// ---- Data types/TPlateData.TcDUT
{attribute 'pack_mode' := '1'}
TYPE TPlateData :
STRUCT
	lrHeight					: LREAL;
	lrEdge					: LREAL;
	alrPartOnPlate			: ARRAY[0..C_MAX_NB_OF_PARTS_ON_PLATE] OF TPositionXY;
	iNbPartOnPlate			: INT;
	alrTakePlatePos			: TPositionXY;
	lrRejectCorrectionY		: LREAL;
	bUseVisionForDrop		: BOOL;
END_STRUCT
END_TYPE

// ---- Data types/TPlatePartStatus.TcDUT
TYPE TPlatePartStatus :
	(
		PPS_Undefined := 0,
		PPS_Present,
		PPS_Absent,
		PPS_BadPart
	);
END_TYPE

// ---- Data types/TPositionXY.TcDUT
{attribute 'pack_mode' := '1'}
TYPE TPositionXY :
STRUCT
	lrX		: LREAL;
	lrY		: LREAL;
END_STRUCT
END_TYPE

// ---- Data types/TPositionXYTheta.TcDUT
{attribute 'pack_mode' := '1'}
TYPE TPositionXYTheta :
STRUCT
	lrX		: LREAL;
	lrY		: LREAL;
	lrTheta	: LREAL;
END_STRUCT
END_TYPE

// ---- Data types/TProbingArea.TcDUT
TYPE TProbingArea :
	(
		PA_BeforeSharpen := 0,
		PA_AfterSharpen,
		PA_WeightCalibration,
		PA_PartLayering1Offset0,
		PA_PartLayering1Offset1,
		PA_PartLayering2Offset0,
		PA_PartLayering2Offset1,
		PA_PartLayering3Offset0,
		PA_PartLayering3Offset1,
		PA_PartLayering4Offset0,
		PA_PartLayering4Offset1,
		PA_END
	);
END_TYPE

// ---- Data types/TProbingLog.TcDUT
{attribute 'pack_mode' := '1'}
TYPE TProbingLog :
STRUCT
	bNewLog					: BOOL;
	eProbingArea				: TProbingArea;
	alrProbingPos				: ARRAY[0..1] OF LREAL;
	iProbingThreshold				: INT;
	iPreviousProbingThreshold		: INT;
END_STRUCT
END_TYPE

// ---- Data types/TprodCounter.TcDUT
{attribute 'pack_mode' := '1'}
TYPE TprodCounter :
STRUCT
	dTotal		:DWORD;
	dGood		:DWORD;
END_STRUCT
END_TYPE

// ---- Data types/TProductionCmd.TcDUT
{attribute 'pack_mode' := '1'}
TYPE TProductionCmd :
STRUCT
	TRequestSample		: TManButton;
	TAutoSampling		: TAutoSampling;
END_STRUCT
END_TYPE

// ---- Data types/TProductionLot.TcDUT
{attribute 'pack_mode' := '1'}
TYPE TProductionLot :
STRUCT
	dLotQty					: DWORD;
	dProdQty				: DWORD;
	dGoodQty				: DWORD;
	dLoadedQty				: DWORD;
	dEstimatedPartTime		: DWORD;
	dEstimatedTimeLeft		: DWORD;
	dProductionTime			: DWORD;
END_STRUCT
END_TYPE

// ---- Data types/TProductionStats.TcDUT
{attribute 'pack_mode' := '1'}
TYPE TProductionStats :
STRUCT
	rQualityRate			: REAL;
	rEfficiencyRate		: REAL;
	rAvailabilityRate		: REAL;
END_STRUCT
END_TYPE

// ---- Data types/TRejectReason.TcDUT
TYPE TRejectReason :
	(
		RR_NoReason:=0,
		RR_PearlingSusHead1,
		RR_PearlingSusHead2,
		RR_PearlingSousHead1,
		RR_PearlingSousHead2
	);
END_TYPE

// ---- Data types/TRejectStatus.TcDUT
TYPE TRejectStatus :
	(
		RS_Ready := 0,
		RS_Locked,
		RS_Empty,
		RS_OpenDrawer
	);
END_TYPE

// ---- Data types/TRobotPos.TcDUT
{attribute 'pack_mode' := '1'}
TYPE TRobotPos :
STRUCT
	X		: LREAL;
	Y		: LREAL;
	Z		: LREAL;
	Theta	: LREAL;
END_STRUCT
END_TYPE

// ---- Data types/TRunCmdBarrel.TcDUT
TYPE TRunCmdBarrel :
	(
		RCB_None,
		RCB_GiveStick,
		RCB_PrepareStick
	);
END_TYPE

// ---- Data types/TRunCmdLift.TcDUT
TYPE TRunCmdLift :
	(
		RCL_None,
		RCL_MoveToPlate,
		RCL_MoveToLoadPlate,
		RCL_MoveToOpenDrawer
	);
END_TYPE

// ---- Data types/TRunCmdLoader.TcDUT
TYPE TRunCmdLoader :
	(
		RCLo_None,
		RCLo_TakePart,
		RCLo_GivePart,
		RCLo_TakePlate,
		RCLo_GivePlate,
		RCLo_Cleaning,
		RCLo_PrepareTakePart,
		RCLo_PrepareDropPart,
		RCLo_MoveToSafe,
		RCLo_SwitchPlate,
		RCLo_EndOfRecipe,
		RCLo_ScanPlate
	);
END_TYPE

// ---- Data types/TRunCmdPearling.TcDUT
TYPE TRunCmdPearling :
	(
		RCP_None,
		RCP_Pearl,
		RCP_ChangeChuck,
		RCP_CheckSharpen
	);
END_TYPE

// ---- Data types/TRunCmdReject.TcDUT
TYPE TRunCmdReject :
	(
		RCR_None,
		RCR_OpenDrawer,
		RCR_LockDrawer,
		RCR_UnlockDrawer
	);
END_TYPE

// ---- Data types/TRunCmdSharpen.TcDUT
TYPE TRunCmdSharpen :
	(
		RCS_None,
		RCS_MoveStep
	);
END_TYPE

// ---- Data types/TRunCmdTable.TcDUT
TYPE TRunCmdTable :
	(
		RCT_None,
		RCT_TakePart,
		RCT_GivePart,
		RCT_Turn,
		RCT_Clean,
		RCT_TurnAndClean
	);
END_TYPE

// ---- Data types/TRunCmdTurnOver.TcDUT
TYPE TRunCmdTurnOver :
	(
		RCTO_None,
		RCTO_TakePart,
		RCTO_GivePart,
		RCTO_Turn
	);
END_TYPE

// ---- Data types/TRunCmdVision.TcDUT
TYPE TRunCmdVision :
	(
		RCV_None,
		RCV_GrabImage,
		RCV_AnalyseImage
	);
END_TYPE

// ---- Data types/TRunData.TcDUT
{attribute 'pack_mode' := '1'}
TYPE TRunData :
STRUCT
	sStatusBarrel			: TRunStatus;
	sStatusLift1			: TRunStatus;
	sStatusLift2			: TRunStatus;
	sStatusLoader		: TRunStatus;
	sStatusPearling		: TRunStatus;
	sStatusReject			: TRunStatus;
	sStatusSharpen		: TRunStatus;
	sStatusTable			: TRunStatus;
	sStatusTurnOver		: TRunStatus;
	sStatusVision			: TRunStatus;
	eCmdBarrel			: TRunCmdBarrel;
	eCmdLift1			: TRunCmdLift;
	eCmdLift2			: TRunCmdLift;
	eCmdLoader			: TRunCmdLoader;
	eCmdPearling		: TRunCmdPearling;
	eCmdReject			: TRunCmdReject;
	eCmdSharpen		: TRunCmdSharpen;
	eCmdTable			: TRunCmdTable;
	eCmdTurnOver		: TRunCmdTurnOver;
	eCmdVision			: TRunCmdVision;
	TDataPearling		: TRunDataPearling;
	TDataTable			: TRunDataTable;
	TDataTurnOver		: TRunDataTurnOver;
	TDataLift1			: TRunDataLift;
	TDataLift2			: TRunDataLift;
	TDataVision			: TRunDataVision;
	TDataReject			: TRunDataReject;
	TDataLoader			: TRunDataLoader;
END_STRUCT
END_TYPE

// ---- Data types/TRunDataLift.TcDUT
{attribute 'pack_mode' := '1'}
TYPE TRunDataLift :
STRUCT
	eLiftPos			: TLiftPos;
END_STRUCT
END_TYPE

// ---- Data types/TRunDataLoader.TcDUT
{attribute 'pack_mode' := '1'}
TYPE TRunDataLoader :
STRUCT
	eTaker				: TLoaderHead;
	eModule				: TLoaderModulePos;
	iLayringPos			: INT;
	iLayringOffsetPos		: INT;
	aTPartData			: ARRAY[0..1] OF TPartData;  (* TLoaderHead *)
	bPlatePresent		: BOOL;
	lrZPositionTakeGive	: LREAL;
	iScanModel			: INT;
	iCurrentScanOK		: INT;
	iCurrentScanTotal		: INT;
END_STRUCT
END_TYPE

// ---- Data types/TRunDataPearling.TcDUT
{attribute 'pack_mode' := '1'}
TYPE TRunDataPearling :
STRUCT
		abUseSpindle				: ARRAY[0..1] OF BOOL;
		sPearlingData				: TPearlingDataHead;
		iLayringPos					: INT;
		iLayringOffsetPos				: INT;
		apsPartData					: ARRAY[0..1] OF POINTER TO TPartData;
		bForceSharpenAfterPearling	: BOOL;
END_STRUCT
END_TYPE

// ---- Data types/TRunDataPlate.TcDUT
{attribute 'pack_mode' := '1'}
TYPE TRunDataPlate :
STRUCT
	ePartStatus	: TPlatePartStatus;
END_STRUCT
END_TYPE

// ---- Data types/TRunDataReject.TcDUT
{attribute 'pack_mode' := '1'}
TYPE TRunDataReject :
STRUCT
	eRejectStatus		: TRejectStatus;
END_STRUCT
END_TYPE

// ---- Data types/TRunDataTable.TcDUT
{attribute 'pack_mode' := '1'}
TYPE TRunDataTable :
STRUCT
	aTPartData						: ARRAY[0..1,0..1,0..1] OF TPartData;	(*Layering, Layering Offset, Side *)
	iGiveTakeLayeringPosition			: INT;
	iGiveTakeLayeringOffsetPosition	: INT;
	eTableSide						: TTableSide;
END_STRUCT
END_TYPE

// ---- Data types/TRunDataTurnOver.TcDUT
{attribute 'pack_mode' := '1'}
TYPE TRunDataTurnOver :
STRUCT
	aTPartData						: ARRAY[0..1] OF TPartData;
END_STRUCT
END_TYPE

// ---- Data types/TRunDataVision.TcDUT
{attribute 'pack_mode' := '1'}
TYPE TRunDataVision :
STRUCT
		iUseModel		: INT;
		iMaxModel		: INT;
		TVisionPartData	: TVisionPartData;
END_STRUCT
END_TYPE

// ---- Data types/TRunStatus.TcDUT
TYPE TRunStatus :
	(
		RS_WaitRequest,
		RS_ProcessRequest1,
		RS_ProcessRequest2,
		RS_NotRunning
	);
END_TYPE

// ---- Data types/TStationGiversTakers.TcDUT
{attribute 'pack_mode' := '1'}
TYPE TStationGiversTakers :
	STRUCT
		(* For  loader *)
		sLoaderTurnOverTakerIn		: TTaker;
		sLoaderTurnOverGiverIn		: TGiver;
		sLoaderTurnOverTakerOut		: TTaker;
		sLoaderTurnOverGiverOut		: TGiver;

		sLoaderTableTakerIn			: TTaker;
		sLoaderTableGiverIn			: TGiver;
		sLoaderTableTakerOut		: TTaker;
		sLoaderTableGiverOut			: TGiver;


		(* For pearling station *)
		sPearlingTakeFromBarrel		:TTaker;

		(* For  barrel *)
		sBarrelGiveToPearling			:TGiver;

	END_STRUCT
END_TYPE

// ---- Data types/TStationIndex.TcDUT
TYPE TStationIndex :
	(SI_LeftLoader:=0, SI_RightLoader,SI_LeftTable,SI_LeftPearling,SI_RightTable,SI_RightPearling,SI_TurnOver,SI_LeftSharpen,SI_RightSharpen,SI_LeftBarrel,SI_RightBarrel,SI_Other);
END_TYPE

// ---- Data types/TStickData.TcDUT
{attribute 'pack_mode' := '1'}
TYPE TStickData :
STRUCT
	iBarrelPos			: INT := -1;
	lrDiameter			: LREAL;
	lrOutLength			: LREAL;
	lrTotalLength			: LREAL;
END_STRUCT
END_TYPE

// ---- Data types/TStickDataMMI.TcDUT
{attribute 'pack_mode' := '1'}
TYPE TStickDataMMI :
STRUCT
	iCompenseWeight				: INT;
	lrMCRCorrectionStep			: LREAL;
	lrMA2MMFactor				: LREAL;
	lrMCRRatio					: LREAL;
END_STRUCT
END_TYPE

// ---- Data types/TStickDataMMIShared.TcDUT
{attribute 'pack_mode' := '1'}
TYPE TStickDataMMIShared :
STRUCT
	iNbOfFwBwSharpen			: INT;
	iNbOfFwBwBeforeTapeMove	: INT;
	lrSharpenSpeed				: LREAL;
	lrSharpenHeight				: LREAL;
	bRestartBeginOfArea			: BOOL;
	lrMinHoldLength				: LREAL;
	bStopOnVacuumLoss			: BOOL;
	bStopOnStickBreak			: BOOL;
	iMCRSharpenSpeed			: INT;
	iWeightTolerance				: INT;
	bStopOnWeightOutOfTolerance	: BOOL;
END_STRUCT
END_TYPE

// ---- Data types/TStickDataShared.TcDUT
{attribute 'pack_mode' := '1'}
TYPE TStickDataShared :
STRUCT
	sStickDataMMIShared		: TStickDataMMIShared;
END_STRUCT
END_TYPE

// ---- Data types/TTableSide.TcDUT
TYPE TTableSide :
	(
		TS_A := 0,
		TS_B,
		TS_Moving
	);
END_TYPE

// ---- Data types/TTaker.TcDUT
{attribute 'pack_mode' := '1'}
TYPE TTaker :
	STRUCT
		bReadyToTake	: BOOL;		(* The taker is ready to take the part *)
		bHasTaken		: BOOL;		(* Part has been taken *)
		bHasNotTaken	: BOOL;		(* Part has not been taken *)
	END_STRUCT
END_TYPE

// ---- Data types/TTransferIndex.TcDUT
TYPE TTransferIndex :
	(TI_Loader:=0,TI_LoaderTableL1,TI_LoaderTableL2,TI_LoaderTableR1,TI_LoaderTableR2,TI_PearlingTableL,TI_PearlingTableR,TI_PearlingTable, TI_LoaderTurnOver,TI_END);
END_TYPE

// ---- Data types/TTurnOverPos.TcDUT
TYPE TTurnOverPos :
	(
		TO_Arm := 0,
		TO_Fix
	);
END_TYPE

// ---- Data types/TVaccumSettings.TcDUT
{attribute 'pack_mode' := '1'}
TYPE TVaccumSettings :
STRUCT
	iBlowing				: INT;
	iWaitWhenVacuumOk	: INT;
	iErrorDelay			: INT;
END_STRUCT
END_TYPE

// ---- Data types/TVacuumSettingsMMI.TcDUT
{attribute 'pack_mode' := '1'}
TYPE TVacuumSettingsMMI :
STRUCT
	TTable				: TVaccumSettings;
	TLoaderHead		: TVaccumSettings;
	TLoaderPlate			: TVaccumSettings;
	TTurnOver			: TVaccumSettings;
	iTablePartialDelay	: INT;
END_STRUCT
END_TYPE

// ---- Data types/TVisionData.TcDUT
{attribute 'pack_mode' := '1'}
TYPE TVisionData :
	STRUCT
		eRequest			: TVisionRequest;
		bRequestDone		: BOOL;
		bRequestError		: BOOL;
		iMajorVersion		: INT;
		iMinorVersion		: INT;
		bAlive				: BOOL;
		bConnected			: BOOL;
		acRefFileName		: STRING(20);
		TPartData			: TVisionPartData;
		bReady				: BOOL;
		bSimRecipe			: BOOL;
		iUseModel			: INT;
		iMaxModel			: INT;
		bMondemaMode		: BOOL;
		bConfigMode			: BOOL;
	END_STRUCT
END_TYPE

// ---- Data types/TVisionPartData.TcDUT
{attribute 'pack_mode' := '1'}
TYPE TVisionPartData :
	STRUCT
		lrX				: LREAL;
		lrY				: LREAL;
		lrTheta			: LREAL;
		lrScore			: LREAL;
		bValid			: BOOL;
		bPresent			: BOOL;
		bImageGrabbed	: BOOL;
	END_STRUCT
END_TYPE

// ---- Data types/TVisionRequest.TcDUT
TYPE TVisionRequest :
	(	VR_None := 0,
		VR_Init,
		VR_Analyse,
		VR_GrabImage
	);
END_TYPE

// ---- Global Variables/Global_Variables.TcGVL
{attribute 'Tc2GvlVarNames'}
(*-----------------------------------------------------------------------------------------------------------------------------------------------------------------------------------------------------------------------------------------------------------------------------------------------------------------------
  GLOBAL CONFIGURATION SPECIFIC TO SOLD MACHINE
 *)
VAR_GLOBAL PERSISTENT
	bUseMDEOption							: BOOL							:= TRUE;	(* MDE option for ETA *)
	bUseRTPOption							: BOOL							:= FALSE;	(* REAL-TIME pearling screen option *)
	bUseTurnOverOption						: BOOL							:= FALSE;	(* TurnOver module is fitted *)
	bUseASOption							: BOOL							:= FALSE;	(* Auto-Sampling screen option *)
	bUseNewBarrelFunction					: BOOL							:= TRUE;	(* Specific function to use 1-4 sectors for each gripper *)
	bUse103059Kludges						: BOOL							:= FALSE;	(* Specific to Blancpain to correct mechanical issues *)
	bRejectPartWithVacuumErrorOnTable		: BOOL							:= FALSE;	(* Try to reject a part if vacuum on table was bad when dropping from loader *)
	bUseFullTapeWidth						: BOOL							:= FALSE;	(* Use full tape width, half for roughing, other half for finish *)
	bUsePearlMoveToSafe						: BOOL							:= FALSE;	(* Use the feature to not move to preref between pearls to save time *)
	bUseLockPlate							: bool							:= False; 	(* Use the lock plate option of the Lifts *)
(* Optimisations *)
	bUse103171OptimA1						: BOOL							:= FALSE;	(* Specific optimisation specified in document 502004-3TC-0001-07 *)
	bUse103171OptimB3						: BOOL							:= FALSE;	(* Specific optimisation specified in document 502004-3TC-0001-07 *)
	bUse103171OptimB5PreMoveXY				: BOOL							:= FALSE;	(* Specific optimisation specified in document 502004-3TC-0001-07 : Pre-move XY to safe when waiting for others *)
	bUse103171OptimB5MoveOnPreSafeZ			: BOOL							:= FALSE;	(* Specific optimisation specified in document 502004-3TC-0001-07 : Say Z in safe if near by safe position even if not in position *)
	bUse103171OptimB5CleanOnBothSide		: BOOL							:= FALSE;	(* Specific optimisation specified in document 502004-3TC-0001-07 : Clean on both side *)
	bUse103171OptimB5CleanOn1Move			: BOOL							:= FALSE;	(* Specific optimisation specified in document 502004-3TC-0001-07 : Clean only on 1 move (no return back *)
END_VAR
VAR_GLOBAL CONSTANT
	C_MAX_NB_OF_ERRORS						: INT							:= 159;		(* 160 errors *)
	C_MAX_NB_OF_PARTS_ON_PLATE				: INT							:= 99;		(* Max nb of parts on plate : 100*)
	C_MAX_NB_OF_PEARLS						: INT							:= 600;		(* Max NB of pearls on 1 side and 1 diameter *)
	C_NB_OF_COM								: INT							:=1;		(* Nb of serial ports *)
	C_COM_NUMBERS							: ARRAY[1..C_NB_OF_COM] OF INT	:= [1];		(* List of serial ports com numbers *)
	C_WEIGHT_TABLE_MAX						: INT							:=25;		(* Nb of point for weight calibration *)
	C_PROD_MODE_GOOD_PART					: BOOL							:= FALSE;	(* False -> Prod quantity is the number of parts on the lift / True -> Prod quantity is the good produced part *)
END_VAR
(*-----------------------------------------------------------------------------------------------------------------------------------------------------------------------------------------------------------------------------------------------------------------------------------------------------------------------*)
VAR_GLOBAL
(* For MDE *)
	{attribute 'OPC.UA.DA' := '1'}
  	{attribute 'OPC.UA.DA.StructuredType' := '1'}
	TMDEData								: TMDE; 									(* TMDE Data *)
(* Internal data *)
	RxBuffer_MCR							: ARRAY[1..C_NB_OF_COM] OF ComBuffer;		(* Reception buffer for MCR *)
	TxBuffer_MCR							: ARRAY[1..C_NB_OF_COM] OF ComBuffer;		(* Transmission buffer for MCR *)
(* Digital IOs *)
	(* Twinsafe *)
	IbV1PowerIsOff					AT %I*	: BOOL;										(* TWINSAFE : Power V1 is off *)
	IbDrivesAreOFF					AT %I*	: BOOL;										(* TWINSAFE : Power on drives is off *)
	IbNoEmergencyStop				AT %I*	: BOOL;										(* TWINSAFE : Emergency stop not pressed *)
	QbStartSafety					AT %Q*	: BOOL;										(* TWINSAFE : Start the safety **Always set to true** *)
	QbPowerOnDrives					AT %Q*	: BOOL;										(* TWINSAFE : Power on drives **Always set to true** *)
	QbResetSafety					AT %Q*	: BOOL;										(* TWINSAFE : Reset the safety errors *)
	(* Doors *)
	IbPearlingDoorsClosed			AT %I*	: BOOL;										(* Pearling doors are closed *)
	IbPearlingDoorsLocked			AT %I*	: BOOL;										(* Pearling doors are locked *)
	IbLoaderDoorsClosed				AT %I*	: BOOL;										(* Loader doors are closed *)
	IbLoaderDoorsLocked				AT %I*	: BOOL;										(* Loader doors are locked *)
	QbLockPearlingDoors				AT %Q*	: BOOL;										(* Lock door on pearling *)
	QbLockLoaderDoors				AT %Q*	: BOOL;										(* Lock door on loader *)
	(* Power supplies *)
	Ib24VOK							AT %I*	: BOOL;										(* 24V power supplies are OK *)
	Ib48VOK							AT %I*	: BOOL;										(* 48V power supplies are OK *)
	(* Light Tower *)
	QbGreenLight					AT %Q*	: BOOL;										(* Green light *)
	QbRedLight						AT %Q*	: BOOL;										(* Red light *)
	QbBlueLight						AT %Q*	: BOOL;										(* Yellow light *)
	(*Air pressure *)
	IbAirPressureOK					AT %I*	: BOOL;										(* Air pressure is OK *)
	(* Vacuum *)
	IbVacuumPumpIsOn				AT %I*	: BOOL;										(* Vacuum pump is powered *)
	IbMainVacuumOK					AT %I*	: BOOL;										(* main vacuum is OK *)
	QbVacuumPumpOn					AT %Q*	: BOOL;										(* Activate vacuum pump *)
	(* Aspiration *)
	IbAspirationIsOn				AT %I*	: BOOL;										(* Aspiration is powered *)
	IbAspirationOK					AT %I*	: BOOL;										(* Aspiration is OK *)
	QbAspirationOn					AT %Q*	: BOOL;										(* Activate aspirator *)
	(* Lift 1 *)
	IbLift1Home						AT %I*	: BOOL;										(* Lift 1 is at home *)
	IbLift1PosLimit					AT %I*	: BOOL;										(* Lift 1 is not down *)
	IbLift1NegLimit					AT %I*	: BOOL;										(* Lift 1 is not up *)
	IbLift1PlateInPos				AT %I*	: BOOL;										(* Plate on lift 1 is in position *)
	IbLift1DrawerInPos				AT %I*	: BOOL;										(* Drawer of lift 1 is in position *)
	IbLift1DrawerLocked				AT %I*	: BOOL;										(* Drawer of lift 1 is locked *)
	IbLift1DrawerUnlocked			AT %I*	: BOOL;										(* Drawer of lift 1 is unlocked *)
	IbLift1PlateLocked				AT %I*	: BOOL;										(* Lift 1 plate is locked *)
	IbLift1PlateUnlocked			AT %I*	: BOOL;										(* Lift 1 plate is unlocked *)
	QbLift1BlueLight				AT %Q*	: BOOL;										(* Blue light for left lift *)
	QbLift1LockPlate				AT %Q*	: BOOL;										(* Lock plate of lift 1 *)
	QbLift1UnlockPlate				AT %Q*	: BOOL;										(* Unlock plate of lift 1 *)
	QbLift1LockDrawer				AT %Q*	: BOOL;										(* Lock drawer of lift 1 *)
	QbLift1UnlockDrawer				AT %Q*	: BOOL;										(* Unlock drawer of lift 1 *)
	(* Lift 2 *)
	IbLift2Home						AT %I*	: BOOL;										(* Lift 1 is at home *)
	IbLift2PosLimit					AT %I*	: BOOL;										(* Lift 2 is not down *)
	IbLift2NegLimit					AT %I*	: BOOL;										(* Lift 2 is not up *)
	IbLift2PlateInPos				AT %I*	: BOOL;										(* Plate on lift 2 is in position *)
	IbLift2DrawerInPos				AT %I*	: BOOL;										(* Drawer of lift 2 is in position *)
	IbLift2DrawerLocked				AT %I*	: BOOL;										(* Drawer of lift 2 is locked *)
	IbLift2DrawerUnlocked			AT %I*	: BOOL;										(* Drawer of lift 2 is unlocked *)
	IbLift2PlateLocked				AT %I*	: BOOL;										(* Lift 2 plate is locked *)
	IbLift2PlateUnlocked			AT %I*	: BOOL;										(* Lift 2 plate is unlocked *)
	QbLift2BlueLight				AT %Q*	: BOOL;										(* Blue light for right lift *)
	QbLift2LockPlate				AT %Q*	: BOOL;										(* Lock plate of lift 2 *)
	QbLift2UnlockPlate				AT %Q*	: BOOL;										(* Unlock plate of lift 2 *)
	QbLift2LockDrawer				AT %Q*	: BOOL;										(* Lock drawer of lift 2 *)
	QbLift2UnlockDrawer				AT %Q*	: BOOL;										(* Unlock drawer of lift 2 *)
	(* Reject *)
	IbRejectPlateInPos				AT %I*	: BOOL;										(* Plate on reject is in position *)
	IbRejectDrawerInPos				AT %I*	: BOOL;										(* Drawer for reject is in position *)
	QbRejectBlueLight				AT %Q*	: BOOL;										(* Blue light for reject *)
	(* Loader *)
	ILoaderMotorXYStatus			AT %I*	: WORD;										(* Digital inputs from loader XY drive *)
	IbLoaderHomeZ1					AT %I*	: BOOL;										(* Home for Head 1 Z axis *)
	IbLoaderPosLimitZ1				AT %I*	: BOOL;										(* Pos. llimit for Head 1 Z axis *)
	IbLoaderNegLimitZ1				AT %I*	: BOOL;										(* Neg. llimit for Head 1 Z axis *)
	IbLoaderHomeZ2					AT %I*	: BOOL;										(* Home for Head 2 Z axis *)
	IbLoaderPosLimitZ2				AT %I*	: BOOL;										(* Pos. llimit for Head 2 Z axis *)
	IbLoaderNegLimitZ2				AT %I*	: BOOL;										(* Neg. llimit for Head 2 Z axis *)
	IbLoaderPlateTakerIsUp			AT %I*	: BOOL;										(* Plate taker is up *)
	IbLoaderPlateTakerIsDown		AT %I*	: BOOL;										(* Plate taker is down *)
	IiLoaderHead1Vacuum				AT %I*	: INT;										(* Vacuum flow on head 1 *)
	IiLoaderHead2Vacuum				AT %I*	: INT;										(* Vacuum flow on head 2 *)
	IbLoaderPlateVacuumOK			AT %I*	: BOOL;										(* Vacuum on plate is OK *)
	ILoaderPlateDistance			AT %I*	: INT;										(* Distance from head to plate *)
	QbLoaderActivateHead1Vacuum		AT %Q*	: BOOL;										(* Activate Head 1 vacuum *)
	QbLoaderActivateHead1Blowing	AT %Q*	: BOOL;										(* Activate Head 1 blowing *)
	QbLoaderActivateHead2Vacuum		AT %Q*	: BOOL;										(* Activate Head 2 vacuum *)
	QbLoaderActivateHead2Blowing	AT %Q*	: BOOL;										(* Activate Head 2 blowing *)
	QbLoaderActivatePlateVacuum		AT %Q*	: BOOL;										(* Activate plate vacuum *)
	QbLoaderActivatePlateBlowing	AT %Q*	: BOOL;										(* Activate plate blowing *)
	QbLoaderPlateTakerDown			AT %Q*	: BOOL;										(* Move down the plate taker part *)
	QbLoaderPlateTakerUp			AT %Q*	: BOOL;										(* Move up the plate taker part *)
	QbLoaderBrushAspirationVacuum	AT %Q*	: BOOL;										(* Activate aspiration on cleaning brush *)
	QbLoaderBrushAspirationBlowing	AT %Q*	: BOOL;										(* Deactivate aspiration on cleaning brush *)
	(* Table *)
	IbTableHome						AT %I*	: BOOL;										(* Home for rotation axis *)
	IbTableLocked					AT %I*	: BOOL;										(* Table is locked in position *)
	IbTableNotLocked				AT %I*	: BOOL;										(* Table is not locked in position *)
	IiTableVacuumPos1Flow			AT %I*	: INT;										(* Vacuum flow on position 1 *)
	IiTableVacuumPos2Flow			AT %I*	: INT;										(* Vacuum flow on position 2 *)
	IiTableVacuumPos3Flow			AT %I*	: INT;										(* Vacuum flow on position 3 *)
	IiTableVacuumPos4Flow			AT %I*	: INT;										(* Vacuum flow on position 4 *)
	IbTableAspirationIsUp			AT %I*	: BOOL;										(* Aspiration module is up *)
	IbTableAspirationIsDown			AT %I*	: BOOL;										(* Aspiration module is down *)
	IbTableCleanBrushIsUp			AT %I*	: BOOL;										(* Clean brush is up *)
	IbTableCleanBrushIsDown			AT %I*	: BOOL;										(* Clean brush is down *)
	QbTableLock						AT %Q*	: BOOL;										(* Lock the table in position *)
	QbTableActivateVacuumPos1		AT %Q*	: BOOL;										(* Activate vacuum on position 1 *)
	QbTableActivateBlowingPos1		AT %Q*	: BOOL;										(* Activate blowing on position 1 *)
	QbTableActivateVacuumPos2		AT %Q*	: BOOL;										(* Activate vacuum on position 2 *)
	QbTableActivateBlowingPos2		AT %Q*	: BOOL;										(* Activate blowing on position 2 *)
	QbTableActivateVacuumPos3		AT %Q*	: BOOL;										(* Activate vacuum on position 3 *)
	QbTableActivateBlowingPos3		AT %Q*	: BOOL;										(* Activate blowing on position 3 *)
	QbTableActivateVacuumPos4		AT %Q*	: BOOL;										(* Activate vacuum on position 4 *)
	QbTableActivateBlowingPos4		AT %Q*	: BOOL;										(* Activate blowing on position 4 *)
	QbTableAspiration13Vacuum		AT %Q*	: BOOL;										(* Activate aspiration on left position *)
	QbTableAspiration13Blowing		AT %Q*	: BOOL;										(* Activate aspiration on right position *)
	QbTableAspiration24Vacuum		AT %Q*	: BOOL;										(* Deactivate aspiration on left position *)
	QbTableAspiration24Blowing		AT %Q*	: BOOL;										(* Deactivate aspiration on right position *)
	QbTableAspirationUp				AT %Q*	: BOOL;										(* Move aspiration module down *)
	QbTableAspirationDown			AT %Q*	: BOOL;										(* Move aspiration module down *)
	QbTableCleanBrushDown			AT %Q*	: BOOL;										(* Move clean brush down *)
	(* Brush *)
	IbBrushHome						AT %I*	: BOOL;										(* Home for Brush axis *)
	IbBrushPosLimit					AT %I*	: BOOL;										(* Pos. llimit for Brush axis *)
	IbBrushNegLimit					AT %I*	: BOOL;										(* Neg limit for Brush axis *)
	QbBrushAspirationVacuum			AT %Q*	: BOOL;										(* Activate aspiration on cleaning brush *)
	QbBrushAspirationBlowing		AT %Q*	: BOOL;										(* Deactivate aspiration on cleaning brush *)
	(* Pearling *)
	IPearlingMotorXYStatus			AT %I*	: WORD;										(* Digital inputs from pearling XY drive *)
	IbPearlingHomeZ1				AT %I*	: BOOL;										(* Home for Z1 axis *)
	IbPearlingPosLimitZ1			AT %I*	: BOOL;										(* Pos. llimit for Z1 axis *)
	IbPearlingNegLimitZ1			AT %I*	: BOOL;										(* Neg. llimit for Z1 axis *)
	IbPearlingHomeZ2				AT %I*	: BOOL;										(* Home for Z2 axis *)
	IbPearlingPosLimitZ2			AT %I*	: BOOL;										(* Pos. llimit for Z2 axis *)
	IbPearlingNegLimitZ2			AT %I*	: BOOL;										(* Neg. llimit for Z2 axis *)
	IbPearlingChuck1Open			AT %I*	: BOOL;										(* Chuck 1 is open *)
	IbPearlingChuck1Closed			AT %I*	: BOOL;										(* Chuck 1 is closed *)
	IbPearlingChuck2Open			AT %I*	: BOOL;										(* Chuck 2 is open *)
	IbPearlingChuck2Closed			AT %I*	: BOOL;										(* Chuck 2 is closed *)
	IbPearlingChangeBroach			AT %I*	: BOOL;										(* Request change broach button*)
	IPearlingContact1Distance		AT %I*	: INT;										(* Distance from sensor to stick 1 contact *)
	IPearlingContact2Distance		AT %I*	: INT;										(* Distance from sensor to stick 2 contact *)
	IPearlingWeightMeasure			AT %I*	: INT;										(* Weight on load sensor *)
	QbPearlingStartMotor1			AT %Q*	: BOOL;										(* Start the pearling 1 motor *)
	QbPearlingStartMotor2			AT %Q*	: BOOL;										(* Start the pearling 2 motor *)
	QbPearlingOpenChuck1			AT %Q*	: BOOL;										(* Open chuck 1 *)
	QbPearlingOpenChuck2			AT %Q*	: BOOL;										(* Open chuck 2 *)
	QbPearlingActivateEject1		AT %Q*	: BOOL;										(* Activate stick 1 ejection *)
	QbPearlingActivateEject2		AT %Q*	: BOOL;										(* Activate stick 2 ejection *)
	QbPearlingActivateBlowing1		AT %Q*	: BOOL;										(* Activate blowing 1 *)
	QbPearlingActivateBlowing2		AT %Q*	: BOOL;										(* Activate blowing 2 *)
	QbPearlingStickLed1				AT %Q*	: BOOL;										(* Stick 1 led is on *)
	QbPearlingStickLed2				AT %Q*	: BOOL;										(* Stick 2 led is on *)
	QbPearlingChangeBroachLight		AT %Q*	: BOOL;										(* Request change broach button light*)
	(* TurnOver *)
	IbTurnOverHome					AT %I*	: BOOL;										(* Home for axis *)
	IbTurnOverArmVacuumOK			AT %I*	: BOOL;										(* Vacuum is OK on arm *)
	IbTurnOverFixVacuumOK			AT %I*	: BOOL;										(* Vacuum is OK on fix position *)
	IbTurnOverFixIsUp				AT %I*	: BOOL;										(* Fix is up *)
	IbTurnOverFixIsDown				AT %I*	: BOOL;										(* Fix is down *)
	QbTurnOverActivateVacuumArm		AT %Q*	: BOOL;										(* Activate vacuum on arm *)
	QbTurnOverActivateBlowingArm	AT %Q*	: BOOL;										(* Activate blowing on arm *)
	QbTurnOverActivateVacuumFix		AT %Q*	: BOOL;										(* Activate vacuum on fix position *)
	QbTurnOverActivateBlowingFix	AT %Q*	: BOOL;										(* Activate blowing on fix position *)
	QbTurnOverMoveFixUp				AT %Q*	: BOOL;										(* Move fix up *)
	QbTurnOverMoveFixDown			AT %Q*	: BOOL;										(* Move fix down *)
	QbTurnOverActivateCleaningBlow	AT %Q*	: BOOL;										(* Activate blowing to clean the holder *)
	(* Sharpen *)
	IbSharpenPosTensioner			AT %I*	: BOOL;										(* The sharpening band is not empty *)
	QbSharpenAspirationVacuum		AT %Q*	: BOOL;										(* Activate aspiration on sharpen*)
	QbSharpenAspirationBlowing		AT %Q*	: BOOL;										(* Deactivate aspiration on sharpen*)
	(* Barrel *)
	IbBarrelStickIsUp				AT %I*	: BOOL;										(* Stick is up *)
	IbBarrelStickIsDown				AT %I*	: BOOL;										(* Stick is down *)
	IbBarrelStickPresent			AT %I*	: BOOL;										(* A stick is present on sensor *)
	IbBarrelIndexed					AT %I*	: BOOL;										(* The barrel is indexed *)
	IbBarrelNotIndexed				AT %I*	: BOOL;										(* The barrel is not indexed *)
	QbBarrelMoveUpStick				AT %Q*	: BOOL;										(* Move up stick *)
	QbBarrelIndexTable				AT %Q*	: BOOL;										(* Move up index *)
	(* Axis *)
	TLoaderXAxis							: AXIS_REF				;					(* linked to loader X axis var in TWINCAT System Manager *)
	TLoaderYAxis							: AXIS_REF;									(* linked to loader Y axis var in TWINCAT System Manager *)
	TLoaderZ1Axis							: AXIS_REF;									(* linked to loader Head 1 Z axis var in TWINCAT System Manager *)
	TLoaderZ2Axis							: AXIS_REF;									(* linked to  loader Head 2 Z axis var in TWINCAT System Manager *)
	TLoaderThetaAxis						: AXIS_REF;									(* linked to  loader Theta axis var in TWINCAT System Manager *)
	TLift1Axis								: AXIS_REF;									(* linked to left lift axis var in TWINCAT System Manager *)
	TLift2Axis								: AXIS_REF;									(* linked to right lift axis var in TWINCAT System Manager *)
	TPearlingXAxis							: AXIS_REF;									(* linked to pearling X axis var in TWINCAT System Manager *)
	TPearlingYAxis							: AXIS_REF;									(* linked to pearling Y axis var in TWINCAT System Manager *)
	TPearlingZ1Axis							: AXIS_REF;									(* linked to pearling Z1 axis var in TWINCAT System Manager *)
	TPearlingZ2Axis							: AXIS_REF;									(* linked to pearling Z2 axis var in TWINCAT System Manager *)
	TTableAxis								: AXIS_REF;									(* linked to table axis var in TWINCAT System Manager *)
	TTurnOverAxis							: AXIS_REF;									(* linked to turn over axis var in TWINCAT System Manager *)
	TSharpenAxis							: AXIS_REF;									(* linked to sharpen axis var in TWINCAT System Manager *)
	TSharpenEncoder							: AXIS_REF;									(* linked to sharpen encoder var in TWINCAT System Manager *)
	TBarrelAxis								: AXIS_REF;									(* linked to barrel axis var in TWINCAT System Manager *)
	TBrushAxis								: AXIS_REF;									(* linked to brush axis var in TWINCAT System Manager *)
END_VAR

// ---- Global Variables/TwinCAT_Configuration.TcGVL
{attribute 'Tc2GvlVarNames'}
(* Generated automatically by TwinCAT - (read only) *)
VAR_CONFIG
	.IbV1PowerIsOff AT %IX52.2 : BOOL;	(*  ~ {LinkedWith:TIID^Device 2 (EtherCAT)^A22.A (Term IO)^A29.4 (TwinSafe IN)^Module 1 (FSOES)^TxPDO^FSOE^PwrV1IsOn_1} *)
	.IbDrivesAreOFF AT %IX52.3 : BOOL;	(*  ~ {LinkedWith:TIID^Device 2 (EtherCAT)^A22.A (Term IO)^A29.4 (TwinSafe IN)^Module 1 (FSOES)^TxPDO^FSOE^DriveIsOn1} *)
	.IbNoEmergencyStop AT %IX52.4 : BOOL;	(*  ~ {LinkedWith:TIID^Device 2 (EtherCAT)^A22.A (Term IO)^A29.1 (TwinSafe PLC)^Module 2 (FSOE)^Standard Out Vars TxPDO 1^Standard Out Var 1} *)
	.QbStartSafety AT %QX0.1 : BOOL;	(*  ~ {LinkedWith:TIID^Device 2 (EtherCAT)^A22.A (Term IO)^A29.1 (TwinSafe PLC)^Module 2 (FSOE)^Standard In Vars RxPDO 1^Standard In Var 1} *)
	.QbPowerOnDrives AT %QX1.1 : BOOL;	(*  ~ {LinkedWith:TIID^Device 2 (EtherCAT)^A22.A (Term IO)^A29.1 (TwinSafe PLC)^Module 2 (FSOE)^Standard In Vars RxPDO 1^Standard In Var 4} *)
	.QbResetSafety AT %QX0.2 : BOOL;	(*  ~ {LinkedWith:TIID^Device 2 (EtherCAT)^A22.A (Term IO)^A29.1 (TwinSafe PLC)^Module 2 (FSOE)^Standard In Vars RxPDO 1^Standard In Var 2;
													TIID^Device 2 (EtherCAT)^A22.A (Term IO)^A29.1 (TwinSafe PLC)^Module 2 (FSOE)^Standard In Vars RxPDO 1^Standard In Var 3;
													TIID^Device 2 (EtherCAT)^A22.A (Term IO)^A29.1 (TwinSafe PLC)^Module 2 (FSOE)^Standard In Vars RxPDO 1^Standard In Var 5} *)
	.IbPearlingDoorsClosed AT %IX52.5 : BOOL;	(*  ~ {LinkedWith:TIID^Device 2 (EtherCAT)^A22.A (Term IO)^A29.3 (TwinSafe IN)^Module 1 (FSOES)^TxPDO^FSOE^Safety3-4Sec1} *)
	.IbPearlingDoorsLocked AT %IX2516.0 : BOOL;	(*  ~ {LinkedWith:TIID^Device 2 (EtherCAT)^A22.A (Term IO)^A29.3 (TwinSafe IN)^Module 1 (FSOES)^TxPDO^FSOE^Safety3-4Sec2} *)
	.IbLoaderDoorsClosed AT %IX52.7 : BOOL;	(*  ~ {LinkedWith:TIID^Device 2 (EtherCAT)^A22.A (Term IO)^A29.3 (TwinSafe IN)^Module 1 (FSOES)^TxPDO^FSOE^Safety1-2Sec1} *)
	.IbLoaderDoorsLocked AT %IX2516.1 : BOOL;	(*  ~ {LinkedWith:TIID^Device 2 (EtherCAT)^A22.A (Term IO)^A29.3 (TwinSafe IN)^Module 1 (FSOES)^TxPDO^FSOE^Safety1-2Sec2} *)
	.QbLockPearlingDoors AT %QX2444.0 : BOOL;	(*  ~ {LinkedWith:TIID^Device 2 (EtherCAT)^A22.A (Term IO)^A26.1^Channel 3^Safety3Lock;TIID^Device 2 (EtherCAT)^A22.A (Term IO)^A26.1^Channel 4^Safety4Lock} *)
	.QbLockLoaderDoors AT %QX2444.1 : BOOL;	(*  ~ {LinkedWith:TIID^Device 2 (EtherCAT)^A22.A (Term IO)^A26.1^Channel 1^Safety1Lock;TIID^Device 2 (EtherCAT)^A22.A (Term IO)^A26.1^Channel 2^Safety2Lock} *)
	.Ib24VOK AT %IX52.0 : BOOL;	(*  ~ {LinkedWith:TIID^Device 2 (EtherCAT)^A22.A (Term IO)^A22.1^Channel 1^Supply24VOn} *)
	.Ib48VOK AT %IX52.1 : BOOL;	(*  ~ {LinkedWith:TIID^Device 2 (EtherCAT)^A22.A (Term IO)^A22.1^Channel 2^Supply48VOn} *)
	.QbGreenLight AT %QX0.3 : BOOL;	(*  ~ {LinkedWith:TIID^Device 2 (EtherCAT)^A22.A (Term IO)^A26.2^Channel 1^GreenLight} *)
	.QbRedLight AT %QX0.5 : BOOL;	(*  ~ {LinkedWith:TIID^Device 2 (EtherCAT)^A22.A (Term IO)^A26.2^Channel 2^RedLight} *)
	.QbBlueLight AT %QX0.4 : BOOL;	(*  ~ {LinkedWith:TIID^Device 2 (EtherCAT)^A22.A (Term IO)^A26.2^Channel 3^BlueLight} *)
	.IbAirPressureOK AT %IX53.1 : BOOL;	(*  ~ {LinkedWith:TIID^Device 2 (EtherCAT)^A22.A (Term IO)^A22.1^Channel 3^AirSupplyOk} *)
	.IbVacuumPumpIsOn AT %IX2516.2 : BOOL;	(*  ~ {LinkedWith:TIID^Device 2 (EtherCAT)^A22.A (Term IO)^A22.1^Channel 6^VacuumPumpIsOn} *)
	.IbMainVacuumOK AT %IX53.3 : BOOL;	(*  ~ {LinkedWith:TIID^Device 2 (EtherCAT)^A22.A (Term IO)^A22.1^Channel 7^VacPumpPressureOk} *)
	.QbVacuumPumpOn AT %QX2444.2 : BOOL;	(*  ~ {LinkedWith:TIID^Device 2 (EtherCAT)^A22.A (Term IO)^A26.2^Channel 5^CmdVacuumPump} *)
	.IbAspirationIsOn AT %IX2524.0 : BOOL;	(*  ~ {LinkedWith:TIID^Device 2 (EtherCAT)^A22.A (Term IO)^A22.2^Channel 2^VacCleanFlowOk} *)
	.IbAspirationOK AT %IX2524.1 : BOOL;	(*  ~ {LinkedWith:TIID^Device 2 (EtherCAT)^A22.A (Term IO)^A22.2^Channel 1^VacuCleanRFiltrOk} *)
	.QbAspirationOn AT %QX2444.3 : BOOL;	(*  ~ {LinkedWith:TIID^Device 2 (EtherCAT)^A22.A (Term IO)^A28.1^Channel 3^VacuCleanRCmd} *)
	.IbLift1Home AT %IX53.5 : BOOL;	(*  ~ {LinkedWith:TIID^Device 2 (EtherCAT)^A31.A (Term Motion)^A31.1 (Lf1CmdMotor)^FB Touch probe status^Touch probe status^Lift1Home} *)
	.IbLift1PosLimit AT %IX2508.0 : BOOL;	(*  ~ {LinkedWith:TIID^Device 2 (EtherCAT)^A22.A (Term IO)^A22.1^Channel 10^Lf1LimiteUp} *)
	.IbLift1NegLimit AT %IX2508.1 : BOOL;	(*  ~ {LinkedWith:TIID^Device 2 (EtherCAT)^A22.A (Term IO)^A22.1^Channel 9^Lf1LimiteDown} *)
	.IbLift1PlateInPos AT %IX54.0 : BOOL;	(*  ~ {LinkedWith:TIID^Device 2 (EtherCAT)^A22.A (Term IO)^A22.1^Channel 11^Lf1PlatelnPos} *)
	.IbLift1DrawerInPos AT %IX54.1 : BOOL;	(*  ~ {LinkedWith:TIID^Device 2 (EtherCAT)^A22.A (Term IO)^A22.1^Channel 12^Lf1DrawInPos} *)
	.QbLift1BlueLight AT %QX1.3 : BOOL;	(*  ~ {LinkedWith:TIID^Device 2 (EtherCAT)^A22.A (Term IO)^A26.2^Channel 6^Lf1BlueLight} *)
	.IbLift2Home AT %IX54.2 : BOOL;	(*  ~ {LinkedWith:TIID^Device 2 (EtherCAT)^A31.A (Term Motion)^A31.2 (Lf2CmdMotor)^FB Touch probe status^Touch probe status^Lift2Home} *)
	.IbLift2PosLimit AT %IX2508.2 : BOOL;	(*  ~ {LinkedWith:TIID^Device 2 (EtherCAT)^A22.A (Term IO)^A22.1^Channel 14^Lf2LimiteUp} *)
	.IbLift2NegLimit AT %IX2508.3 : BOOL;	(*  ~ {LinkedWith:TIID^Device 2 (EtherCAT)^A22.A (Term IO)^A22.1^Channel 13^Lf2LimiteDown} *)
	.IbLift2PlateInPos AT %IX54.5 : BOOL;	(*  ~ {LinkedWith:TIID^Device 2 (EtherCAT)^A22.A (Term IO)^A22.1^Channel 15^Lf2PlatelnPos} *)
	.IbLift2DrawerInPos AT %IX54.6 : BOOL;	(*  ~ {LinkedWith:TIID^Device 2 (EtherCAT)^A22.A (Term IO)^A22.1^Channel 16^Lf2DrawlnPos} *)
	.QbLift2BlueLight AT %QX1.4 : BOOL;	(*  ~ {LinkedWith:TIID^Device 2 (EtherCAT)^A22.A (Term IO)^A26.2^Channel 7^Lf2BlueLight} *)
	.IbRejectPlateInPos AT %IX54.7 : BOOL;	(*  ~ {LinkedWith:TIID^Device 2 (EtherCAT)^A22.A (Term IO)^A22.2^Channel 5^RjPlatelnPos} *)
	.IbRejectDrawerInPos AT %IX55.0 : BOOL;	(*  ~ {LinkedWith:TIID^Device 2 (EtherCAT)^A22.A (Term IO)^A22.2^Channel 6^RjDrawerlnPos} *)
	.QbRejectBlueLight AT %QX1.5 : BOOL;	(*  ~ {LinkedWith:TIID^Device 2 (EtherCAT)^A22.A (Term IO)^A26.2^Channel 9^RjBlueLight} *)
	.ILoaderMotorXYStatus AT %IB2512 : WORD;	(*  ~ {LinkedWith:TIID^Device 2 (EtherCAT)^A17.2 (PoAxMotor PoAyMotor)^AT 1^Digital inputs, state} *)
	.IbLoaderHomeZ1 AT %IX55.3 : BOOL;	(*  ~ {LinkedWith:TIID^Device 2 (EtherCAT)^A31.A (Term Motion)^A33.1 (PoAz1CmdMotor)^STM Status^Status^LoaderZ1Home} *)
	.IbLoaderPosLimitZ1 AT %IX55.4 : BOOL;	(*  ~ {LinkedWith:TIID^Device 2 (EtherCAT)^A22.A (Term IO)^A22.2^Channel 7^PoAz1LimiteDown} *)
	.IbLoaderNegLimitZ1 AT %IX55.5 : BOOL;	(*  ~ {LinkedWith:TIID^Device 2 (EtherCAT)^A22.A (Term IO)^A22.2^Channel 8^PoAz1LimiteUp} *)
	.IbLoaderHomeZ2 AT %IX55.6 : BOOL;	(*  ~ {LinkedWith:TIID^Device 2 (EtherCAT)^A31.A (Term Motion)^A33.2 (PoAz2CmdMotor)^STM Status^Status^LoaderZ2Home} *)
	.IbLoaderPosLimitZ2 AT %IX55.7 : BOOL;	(*  ~ {LinkedWith:TIID^Device 2 (EtherCAT)^A22.A (Term IO)^A22.2^Channel 10^PoAz2LimiteDown} *)
	.IbLoaderNegLimitZ2 AT %IX56.0 : BOOL;	(*  ~ {LinkedWith:TIID^Device 2 (EtherCAT)^A22.A (Term IO)^A22.2^Channel 11^PoAz2LimiteUp} *)
	.IbLoaderPlateTakerIsUp AT %IX56.3 : BOOL;	(*  ~ {LinkedWith:TIID^Device 2 (EtherCAT)^A22.A (Term IO)^A22.2^Channel 13^PoTakPalUp} *)
	.IbLoaderPlateTakerIsDown AT %IX56.4 : BOOL;	(*  ~ {LinkedWith:TIID^Device 2 (EtherCAT)^A22.A (Term IO)^A22.2^Channel 14^PoTakPalDown} *)
	.IbLoaderHead1VacuumOK AT %IX55.1 : BOOL;	(*  ~ {LinkedWith:TIID^Device 2 (EtherCAT)^A22.A (Term IO)^A22.2^Channel 9^PoAz1VacOK} *)
	.IbLoaderHead2VacuumOK AT %IX55.2 : BOOL;	(*  ~ {LinkedWith:TIID^Device 2 (EtherCAT)^A22.A (Term IO)^A22.2^Channel 12^PoAz2VacOK} *)
	.IbLoaderPlateVacuumOK AT %IX56.2 : BOOL;	(*  ~ {LinkedWith:TIID^Device 2 (EtherCAT)^A22.A (Term IO)^A22.2^Channel 15^PoTakPlaVacOK} *)
	.ILoaderPlateDistance AT %IB4 : INT;	(*  ~ {LinkedWith:TIID^Device 2 (EtherCAT)^A22.A (Term IO)^A25.1^AI Standard Channel 1^PoTrayHeigMeas} *)
	.QbLoaderActivateHead1Vacuum AT %QX1.6 : BOOL;	(*  ~ {LinkedWith:TIID^Device 2 (EtherCAT)^A79.1^Byte 0^Output^PoAz1VacOn} *)
	.QbLoaderActivateHead1Blowing AT %QX1.7 : BOOL;	(*  ~ {LinkedWith:TIID^Device 2 (EtherCAT)^A79.1^Byte 0^Output^PoAz1BlowOn} *)
	.QbLoaderActivateHead2Vacuum AT %QX2.0 : BOOL;	(*  ~ {LinkedWith:TIID^Device 2 (EtherCAT)^A79.1^Byte 0^Output^PoAz2VacOn} *)
	.QbLoaderActivateHead2Blowing AT %QX2.1 : BOOL;	(*  ~ {LinkedWith:TIID^Device 2 (EtherCAT)^A79.1^Byte 0^Output^PoAz2BlowOn} *)
	.QbLoaderActivatePlateVacuum AT %QX2.2 : BOOL;	(*  ~ {LinkedWith:TIID^Device 2 (EtherCAT)^A79.1^Byte 1^Output^PoTakPlatVacOn} *)
	.QbLoaderActivatePlateBlowing AT %QX2.3 : BOOL;	(*  ~ {LinkedWith:TIID^Device 2 (EtherCAT)^A79.1^Byte 1^Output^PoTakPlatBlowOn} *)
	.QbLoaderPlateTakerDown AT %QX2.4 : BOOL;	(*  ~ {LinkedWith:TIID^Device 2 (EtherCAT)^A75.1^Byte 1^Output^PoTkPIaGoDown} *)
	.QbLoaderPlateTakerUp AT %QX2.5 : BOOL;	(*  ~ {LinkedWith:TIID^Device 2 (EtherCAT)^A75.1^Byte 1^Output^PoTkPlaGoUp} *)
	.QbLoaderBrushAspirationVacuum AT %QX2448.0 : BOOL;	(*  ~ {LinkedWith:TIID^Device 2 (EtherCAT)^A79.1^Byte 3^Output^AspReOn} *)
	.QbLoaderBrushAspirationBlowing AT %QX2448.1 : BOOL;	(*  ~ {LinkedWith:TIID^Device 2 (EtherCAT)^A79.1^Byte 3^Output^AspReOff} *)
	.IbTableHome AT %IX56.5 : BOOL;	(*  ~ {LinkedWith:TIID^Device 2 (EtherCAT)^A17.3 (RtMotor)^AT^Digital inputs, state} *)
	.IbTableLocked AT %IX56.6 : BOOL;	(*  ~ {LinkedWith:TIID^Device 2 (EtherCAT)^A22.A (Term IO)^A22.3^Channel 13^Rtlndexed} *)
	.IbTableNotLocked AT %IX56.7 : BOOL;	(*  ~ {LinkedWith:TIID^Device 2 (EtherCAT)^A22.A (Term IO)^A22.3^Channel 14^RtUnindexed} *)
	.IiTableVacuumPos1Pressure AT %IB2500 : INT;	(*  ~ {LinkedWith:TIID^Device 2 (EtherCAT)^A22.A (Term IO)^A25.2^AI Standard Channel 1^RtLayring1Vac} *)
	.IiTableVacuumPos2Pressure AT %IB2502 : INT;	(*  ~ {LinkedWith:TIID^Device 2 (EtherCAT)^A22.A (Term IO)^A25.2^AI Standard Channel 2^RtLayring2Vac} *)
	.IiTableVacuumPos3Pressure AT %IB2504 : INT;	(*  ~ {LinkedWith:TIID^Device 2 (EtherCAT)^A22.A (Term IO)^A25.2^AI Standard Channel 3^RtLayring3Vac} *)
	.IiTableVacuumPos4Pressure AT %IB2506 : INT;	(*  ~ {LinkedWith:TIID^Device 2 (EtherCAT)^A22.A (Term IO)^A25.2^AI Standard Channel 4^RtLayring4Vac} *)
	.IbTableAspirationIsUp AT %IX57.4 : BOOL;	(*  ~ {LinkedWith:TIID^Device 2 (EtherCAT)^A22.A (Term IO)^A22.3^Channel 15^RtSpAspIsUp} *)
	.IbTableAspirationIsDown AT %IX57.5 : BOOL;	(*  ~ {LinkedWith:TIID^Device 2 (EtherCAT)^A22.A (Term IO)^A22.3^Channel 16^RtSpinAspIsDown} *)
	.QbTableLock AT %QX2.6 : BOOL;	(*  ~ {LinkedWith:TIID^Device 2 (EtherCAT)^A75.1^Byte 0^Output^RtRlndexCmd} *)
	.QbTableActivateVacuumPos1 AT %QX2.7 : BOOL;	(*  ~ {LinkedWith:TIID^Device 2 (EtherCAT)^A79.1^Byte 0^Output^RtLayring1VacOn} *)
	.QbTableActivateBlowingPos1 AT %QX3.0 : BOOL;	(*  ~ {LinkedWith:TIID^Device 2 (EtherCAT)^A79.1^Byte 0^Output^RtLayring1BlowOn} *)
	.QbTableActivateVacuumPos2 AT %QX3.1 : BOOL;	(*  ~ {LinkedWith:TIID^Device 2 (EtherCAT)^A79.1^Byte 1^Output^RtLayring2VacOn} *)
	.QbTableActivateBlowingPos2 AT %QX3.2 : BOOL;	(*  ~ {LinkedWith:TIID^Device 2 (EtherCAT)^A79.1^Byte 1^Output^RtLayring2BlowOn} *)
	.QbTableActivateVacuumPos3 AT %QX3.3 : BOOL;	(*  ~ {LinkedWith:TIID^Device 2 (EtherCAT)^A79.1^Byte 1^Output^RtLayring3VacOn} *)
	.QbTableActivateBlowingPos3 AT %QX3.4 : BOOL;	(*  ~ {LinkedWith:TIID^Device 2 (EtherCAT)^A79.1^Byte 1^Output^RtLayring3BlowOn} *)
	.QbTableActivateVacuumPos4 AT %QX3.5 : BOOL;	(*  ~ {LinkedWith:TIID^Device 2 (EtherCAT)^A79.1^Byte 1^Output^RtLayring4VacOn} *)
	.QbTableActivateBlowingPos4 AT %QX3.6 : BOOL;	(*  ~ {LinkedWith:TIID^Device 2 (EtherCAT)^A79.1^Byte 1^Output^RtLayring4BlowOn} *)
	.QbTableAspiration13Vacuum AT %QX2448.2 : BOOL;	(*  ~ {LinkedWith:TIID^Device 2 (EtherCAT)^A79.1^Byte 2^Output^AspPe1On} *)
	.QbTableAspiration13Blowing AT %QX2448.3 : BOOL;	(*  ~ {LinkedWith:TIID^Device 2 (EtherCAT)^A79.1^Byte 2^Output^AspPe1Off} *)
	.QbTableAspiration24Vacuum AT %QX2448.4 : BOOL;	(*  ~ {LinkedWith:TIID^Device 2 (EtherCAT)^A79.1^Byte 3^Output^AspPe2On} *)
	.QbTableAspiration24Blowing AT %QX2448.5 : BOOL;	(*  ~ {LinkedWith:TIID^Device 2 (EtherCAT)^A79.1^Byte 3^Output^AspPe2Off} *)
	.QbTableAspirationUp AT %QX4.2 : BOOL;	(*  ~ {LinkedWith:TIID^Device 2 (EtherCAT)^A75.1^Byte 1^Output^RtRSpinAspGoUp} *)
	.QbTableAspirationDown AT %QX4.3 : BOOL;	(*  ~ {LinkedWith:TIID^Device 2 (EtherCAT)^A75.1^Byte 1^Output^RtRSpinAspGoDown} *)
	.IbBrushHome AT %IX2496.0 : BOOL;	(*  ~ {LinkedWith:TIID^Device 2 (EtherCAT)^A22.A (Term IO)^A22.4^Channel 13^BrHomePos} *)
	.IbBrushPosLimit AT %IX2496.1 : BOOL;	(*  ~ {LinkedWith:TIID^Device 2 (EtherCAT)^A22.A (Term IO)^A22.4^Channel 14^BrLimit+} *)
	.IbBrushNegLimit AT %IX2496.2 : BOOL;	(*  ~ {LinkedWith:TIID^Device 2 (EtherCAT)^A22.A (Term IO)^A22.4^Channel 15^BrLimit-} *)
	.QbBrushAspirationVacuum AT %QX2448.6 : BOOL;	(*  ~ {LinkedWith:TIID^Device 2 (EtherCAT)^A79.1^Byte 2^Output^AspMoBrOn} *)
	.QbBrushAspirationBlowing AT %QX2448.7 : BOOL;	(*  ~ {LinkedWith:TIID^Device 2 (EtherCAT)^A79.1^Byte 2^Output^AspMoBrOff} *)
	.IPearlingMotorXYStatus AT %IB2514 : WORD;	(*  ~ {LinkedWith:TIID^Device 2 (EtherCAT)^A17.1 (PeAxMotor PeAyMotor)^AT 1^Digital inputs, state} *)
	.IbPearlingHomeZ1 AT %IX58.1 : BOOL;	(*  ~ {LinkedWith:TIID^Device 2 (EtherCAT)^A22.A (Term IO)^A22.3^Channel 4^PeLAzIsHome} *)
	.IbPearlingPosLimitZ1 AT %IX58.2 : BOOL;	(*  ~ {LinkedWith:TIID^Device 2 (EtherCAT)^A22.A (Term IO)^A22.3^Channel 5^PeLAzLimitUp} *)
	.IbPearlingNegLimitZ1 AT %IX58.3 : BOOL;	(*  ~ {LinkedWith:TIID^Device 2 (EtherCAT)^A22.A (Term IO)^A22.3^Channel 6^PeLAzLimitDown} *)
	.IbPearlingHomeZ2 AT %IX58.4 : BOOL;	(*  ~ {LinkedWith:TIID^Device 2 (EtherCAT)^A22.A (Term IO)^A22.3^Channel 1^PeRAzIsHome} *)
	.IbPearlingPosLimitZ2 AT %IX58.5 : BOOL;	(*  ~ {LinkedWith:TIID^Device 2 (EtherCAT)^A22.A (Term IO)^A22.3^Channel 2^PeRAzLimitUp} *)
	.IbPearlingNegLimitZ2 AT %IX58.6 : BOOL;	(*  ~ {LinkedWith:TIID^Device 2 (EtherCAT)^A22.A (Term IO)^A22.3^Channel 3^PeRAzLimitDown} *)
	.IbPearlingChuck1Open AT %IX58.7 : BOOL;	(*  ~ {LinkedWith:TIID^Device 2 (EtherCAT)^A22.A (Term IO)^A22.3^Channel 10^SpLGripIsOpen} *)
	.IbPearlingChuck1Closed AT %IX59.0 : BOOL;	(*  ~ {LinkedWith:TIID^Device 2 (EtherCAT)^A22.A (Term IO)^A22.3^Channel 9^SpLGripIsClosed} *)
	.IbPearlingChuck2Open AT %IX59.1 : BOOL;	(*  ~ {LinkedWith:TIID^Device 2 (EtherCAT)^A22.A (Term IO)^A22.3^Channel 8^SpRGripIsOpen} *)
	.IbPearlingChuck2Closed AT %IX59.2 : BOOL;	(*  ~ {LinkedWith:TIID^Device 2 (EtherCAT)^A22.A (Term IO)^A22.3^Channel 7^SpRGripIsClosed} *)
	.IbPearlingChangeBroach AT %IX2516.3 : BOOL;	(*  ~ {LinkedWith:TIID^Device 2 (EtherCAT)^A22.A (Term IO)^A22.1^Channel 4^PeSeqChangSpin} *)
	.IPearlingContact1Distance AT %IB6 : INT;	(*  ~ {LinkedWith:TIID^Device 2 (EtherCAT)^A22.A (Term IO)^A25.1^AI Standard Channel 3^PeLAzPresCtrl} *)
	.IPearlingContact2Distance AT %IB8 : INT;	(*  ~ {LinkedWith:TIID^Device 2 (EtherCAT)^A22.A (Term IO)^A25.1^AI Standard Channel 2^PeRAzPresCtrl} *)
	.IPearlingWeightMeasure AT %IB10 : INT;	(*  ~ {LinkedWith:TIID^Device 2 (EtherCAT)^A22.A (Term IO)^A25.3^AI Standard Channel 1^CaLoadSensor} *)
	.QbPearlingStartMotor1 AT %QX4.4 : BOOL;	(*  ~ {LinkedWith:TIID^Device 2 (EtherCAT)^A22.A (Term IO)^A28.1^Channel 2^SpLCtrlMot} *)
	.QbPearlingStartMotor2 AT %QX4.5 : BOOL;	(*  ~ {LinkedWith:TIID^Device 2 (EtherCAT)^A22.A (Term IO)^A28.1^Channel 1^SpRCtrlMot} *)
	.QbPearlingOpenChuck1 AT %QX4.6 : BOOL;	(*  ~ {LinkedWith:TIID^Device 2 (EtherCAT)^A22.A (Term IO)^A26.2^Channel 10^SpLOpenGrip} *)
	.QbPearlingOpenChuck2 AT %QX4.7 : BOOL;	(*  ~ {LinkedWith:TIID^Device 2 (EtherCAT)^A22.A (Term IO)^A26.2^Channel 4^SpROpenGrip} *)
	.QbPearlingActivateEject1 AT %QX5.0 : BOOL;	(*  ~ {LinkedWith:TIID^Device 2 (EtherCAT)^A75.1^Byte 0^Output^SpLPneuEjector} *)
	.QbPearlingActivateEject2 AT %QX5.1 : BOOL;	(*  ~ {LinkedWith:TIID^Device 2 (EtherCAT)^A75.1^Byte 0^Output^SpRPneuEjector} *)
	.QbPearlingActivateBlowing1 AT %QX5.2 : BOOL;	(*  ~ {LinkedWith:TIID^Device 2 (EtherCAT)^A75.1^Byte 0^Output^SpLAirOn} *)
	.QbPearlingActivateBlowing2 AT %QX5.3 : BOOL;	(*  ~ {LinkedWith:TIID^Device 2 (EtherCAT)^A75.1^Byte 0^Output^SpRAirOn} *)
	.QbPearlingStickLed1 AT %QX5.5 : BOOL;	(*  ~ {LinkedWith:TIID^Device 2 (EtherCAT)^A22.A (Term IO)^A26.2^Channel 12^SpLLedApp} *)
	.QbPearlingStickLed2 AT %QX5.6 : BOOL;	(*  ~ {LinkedWith:TIID^Device 2 (EtherCAT)^A22.A (Term IO)^A26.2^Channel 13^SpRLedApp} *)
	.QbPearlingChangeBroachLight AT %QX2444.5 : BOOL;	(*  ~ {LinkedWith:TIID^Device 2 (EtherCAT)^A22.A (Term IO)^A26.2^Channel 11^PeLedSeqChangSp} *)
	.IbTurnOverHome AT %IX59.5 : BOOL;	(*  ~ {LinkedWith:TIID^Device 2 (EtherCAT)^A31.A (Term Motion)^A33.4 (ReCmdMotor)^STM Status^Status^TurnOverHome} *)
	.IbTurnOverArmVacuumOK AT %IX59.6 : BOOL;	(*  ~ {LinkedWith:TIID^Device 2 (EtherCAT)^A22.A (Term IO)^A22.4^Channel 1^ReManipVacOK} *)
	.IbTurnOverFixVacuumOK AT %IX59.7 : BOOL;	(*  ~ {LinkedWith:TIID^Device 2 (EtherCAT)^A22.A (Term IO)^A22.4^Channel 2^ReVacLayringOK} *)
	.IbTurnOverFixIsUp AT %IX60.0 : BOOL;	(*  ~ {LinkedWith:TIID^Device 2 (EtherCAT)^A22.A (Term IO)^A22.4^Channel 4^RelsUp} *)
	.IbTurnOverFixIsDown AT %IX60.1 : BOOL;	(*  ~ {LinkedWith:TIID^Device 2 (EtherCAT)^A22.A (Term IO)^A22.4^Channel 3^RelsDown} *)
	.QbTurnOverActivateVacuumArm AT %QX5.7 : BOOL;	(*  ~ {LinkedWith:TIID^Device 2 (EtherCAT)^A79.1^Byte 0^Output^ReManipVacOn} *)
	.QbTurnOverActivateBlowingArm AT %QX6.0 : BOOL;	(*  ~ {LinkedWith:TIID^Device 2 (EtherCAT)^A79.1^Byte 0^Output^ReManipBlowOn} *)
	.QbTurnOverActivateVacuumFix AT %QX6.1 : BOOL;	(*  ~ {LinkedWith:TIID^Device 2 (EtherCAT)^A79.1^Byte 2^Output^ReLayringVacOn} *)
	.QbTurnOverActivateBlowingFix AT %QX6.2 : BOOL;	(*  ~ {LinkedWith:TIID^Device 2 (EtherCAT)^A79.1^Byte 2^Output^ReLayringBlowOn} *)
	.QbTurnOverMoveFixUp AT %QX6.3 : BOOL;	(*  ~ {LinkedWith:TIID^Device 2 (EtherCAT)^A75.1^Byte 1^Output^ReGoUp} *)
	.QbTurnOverMoveFixDown AT %QX6.4 : BOOL;	(*  ~ {LinkedWith:TIID^Device 2 (EtherCAT)^A75.1^Byte 1^Output^ReGoDown} *)
	.QbTurnOverActivateCleaningBlow AT %QX6.6 : BOOL;	(*  ~ {LinkedWith:TIID^Device 2 (EtherCAT)^A75.1^Byte 0^Output^ReBlowing} *)
	.IbSharpenPosTensioner AT %IX2520.0 : BOOL;	(*  ~ {LinkedWith:TIID^Device 2 (EtherCAT)^A22.A (Term IO)^A22.4^Channel 7^ShCtrlPosTend} *)
	.QbSharpenAspirationVacuum AT %QX2449.0 : BOOL;	(*  ~ {LinkedWith:TIID^Device 2 (EtherCAT)^A79.1^Byte 3^Output^AspAffOn} *)
	.QbSharpenAspirationBlowing AT %QX2449.1 : BOOL;	(*  ~ {LinkedWith:TIID^Device 2 (EtherCAT)^A79.1^Byte 3^Output^AspAffOff} *)
	.IbBarrelStickIsUp AT %IX60.4 : BOOL;	(*  ~ {LinkedWith:TIID^Device 2 (EtherCAT)^A22.A (Term IO)^A22.4^Channel 11^ClSticklsUp} *)
	.IbBarrelStickIsDown AT %IX60.5 : BOOL;	(*  ~ {LinkedWith:TIID^Device 2 (EtherCAT)^A22.A (Term IO)^A22.4^Channel 10^ClSticklsDown} *)
	.IbBarrelStickPresent AT %IX60.6 : BOOL;	(*  ~ {LinkedWith:TIID^Device 2 (EtherCAT)^A22.A (Term IO)^A22.4^Channel 12^ClSticklsPres} *)
	.IbBarrelIndexed AT %IX60.7 : BOOL;	(*  ~ {LinkedWith:TIID^Device 2 (EtherCAT)^A22.A (Term IO)^A22.4^Channel 8^Balndexed} *)
	.IbBarrelNotIndexed AT %IX61.0 : BOOL;	(*  ~ {LinkedWith:TIID^Device 2 (EtherCAT)^A22.A (Term IO)^A22.4^Channel 9^ClNotIndexed} *)
	.QbBarrelMoveUpStick AT %QX7.0 : BOOL;	(*  ~ {LinkedWith:TIID^Device 2 (EtherCAT)^A75.1^Byte 1^Output^BaPushUpStick} *)
	.QbBarrelIndexTable AT %QX7.1 : BOOL;	(*  ~ {LinkedWith:TIID^Device 2 (EtherCAT)^A75.1^Byte 1^Output^CllndexCmd} *)
	.TLoaderXAxis.PlcToNc AT %QB264 : PLCTONC_AXIS_REF;	(*  ~ {LinkedWith:TINC^NC-Task 1 SAF^Axes^Loader X^Entrées^Loader X_FromPlc} *)
	.TLoaderXAxis.NcToPlc AT %IB318 : NCTOPLC_AXIS_REF;	(*  ~ {LinkedWith:TINC^NC-Task 1 SAF^Axes^Loader X^Sorties^Loader X_ToPlc} *)
	.TLoaderYAxis.PlcToNc AT %QB392 : PLCTONC_AXIS_REF;	(*  ~ {LinkedWith:TINC^NC-Task 1 SAF^Axes^Loader Y^Entrées^Loader Y_FromPlc} *)
	.TLoaderYAxis.NcToPlc AT %IB446 : NCTOPLC_AXIS_REF;	(*  ~ {LinkedWith:TINC^NC-Task 1 SAF^Axes^Loader Y^Sorties^Loader Y_ToPlc} *)
	.TLoaderZ1Axis.PlcToNc AT %QB520 : PLCTONC_AXIS_REF;	(*  ~ {LinkedWith:TINC^NC-Task 1 SAF^Axes^Loader Z1^Entrées^Loader Z1_FromPlc} *)
	.TLoaderZ1Axis.NcToPlc AT %IB574 : NCTOPLC_AXIS_REF;	(*  ~ {LinkedWith:TINC^NC-Task 1 SAF^Axes^Loader Z1^Sorties^Loader Z1_ToPlc} *)
	.TLoaderZ2Axis.PlcToNc AT %QB648 : PLCTONC_AXIS_REF;	(*  ~ {LinkedWith:TINC^NC-Task 1 SAF^Axes^Loader Z2^Entrées^Loader Z2_FromPlc} *)
	.TLoaderZ2Axis.NcToPlc AT %IB702 : NCTOPLC_AXIS_REF;	(*  ~ {LinkedWith:TINC^NC-Task 1 SAF^Axes^Loader Z2^Sorties^Loader Z2_ToPlc} *)
	.TLoaderThetaAxis.PlcToNc AT %QB776 : PLCTONC_AXIS_REF;	(*  ~ {LinkedWith:TINC^NC-Task 1 SAF^Axes^Loader Theta^Entrées^Loader Theta_FromPlc} *)
	.TLoaderThetaAxis.NcToPlc AT %IB830 : NCTOPLC_AXIS_REF;	(*  ~ {LinkedWith:TINC^NC-Task 1 SAF^Axes^Loader Theta^Sorties^Loader Theta_ToPlc} *)
	.TLift1Axis.PlcToNc AT %QB904 : PLCTONC_AXIS_REF;	(*  ~ {LinkedWith:TINC^NC-Task 1 SAF^Axes^Lift1^Entrées^Lift1_FromPlc} *)
	.TLift1Axis.NcToPlc AT %IB958 : NCTOPLC_AXIS_REF;	(*  ~ {LinkedWith:TINC^NC-Task 1 SAF^Axes^Lift1^Sorties^Lift1_ToPlc} *)
	.TLift2Axis.PlcToNc AT %QB1032 : PLCTONC_AXIS_REF;	(*  ~ {LinkedWith:TINC^NC-Task 1 SAF^Axes^Lift2^Entrées^Lift2_FromPlc} *)
	.TLift2Axis.NcToPlc AT %IB1086 : NCTOPLC_AXIS_REF;	(*  ~ {LinkedWith:TINC^NC-Task 1 SAF^Axes^Lift2^Sorties^Lift2_ToPlc} *)
	.TPearlingXAxis.PlcToNc AT %QB1160 : PLCTONC_AXIS_REF;	(*  ~ {LinkedWith:TINC^NC-Task 1 SAF^Axes^Pearling X^Entrées^Pearling X_FromPlc} *)
	.TPearlingXAxis.NcToPlc AT %IB1214 : NCTOPLC_AXIS_REF;	(*  ~ {LinkedWith:TINC^NC-Task 1 SAF^Axes^Pearling X^Sorties^Pearling X_ToPlc} *)
	.TPearlingYAxis.PlcToNc AT %QB1288 : PLCTONC_AXIS_REF;	(*  ~ {LinkedWith:TINC^NC-Task 1 SAF^Axes^Pearling Y^Entrées^Pearling Y_FromPlc} *)
	.TPearlingYAxis.NcToPlc AT %IB1342 : NCTOPLC_AXIS_REF;	(*  ~ {LinkedWith:TINC^NC-Task 1 SAF^Axes^Pearling Y^Sorties^Pearling Y_ToPlc} *)
	.TPearlingZ1Axis.PlcToNc AT %QB1416 : PLCTONC_AXIS_REF;	(*  ~ {LinkedWith:TINC^NC-Task 1 SAF^Axes^Pearling Z1^Entrées^Pearling Z1_FromPlc} *)
	.TPearlingZ1Axis.NcToPlc AT %IB1470 : NCTOPLC_AXIS_REF;	(*  ~ {LinkedWith:TINC^NC-Task 1 SAF^Axes^Pearling Z1^Sorties^Pearling Z1_ToPlc} *)
	.TPearlingZ2Axis.PlcToNc AT %QB1544 : PLCTONC_AXIS_REF;	(*  ~ {LinkedWith:TINC^NC-Task 1 SAF^Axes^Pearling Z2^Entrées^Pearling Z2_FromPlc} *)
	.TPearlingZ2Axis.NcToPlc AT %IB1598 : NCTOPLC_AXIS_REF;	(*  ~ {LinkedWith:TINC^NC-Task 1 SAF^Axes^Pearling Z2^Sorties^Pearling Z2_ToPlc} *)
	.TTableAxis.PlcToNc AT %QB1672 : PLCTONC_AXIS_REF;	(*  ~ {LinkedWith:TINC^NC-Task 1 SAF^Axes^Table^Entrées^Table_FromPlc} *)
	.TTableAxis.NcToPlc AT %IB1726 : NCTOPLC_AXIS_REF;	(*  ~ {LinkedWith:TINC^NC-Task 1 SAF^Axes^Table^Sorties^Table_ToPlc} *)
	.TTurnOverAxis.PlcToNc AT %QB1928 : PLCTONC_AXIS_REF;	(*  ~ {LinkedWith:TINC^NC-Task 1 SAF^Axes^TurnOver^Entrées^TurnOver_FromPlc} *)
	.TTurnOverAxis.NcToPlc AT %IB1982 : NCTOPLC_AXIS_REF;	(*  ~ {LinkedWith:TINC^NC-Task 1 SAF^Axes^TurnOver^Sorties^TurnOver_ToPlc} *)
	.TSharpenAxis.PlcToNc AT %QB2056 : PLCTONC_AXIS_REF;	(*  ~ {LinkedWith:TINC^NC-Task 1 SAF^Axes^Sharpen^Entrées^Sharpen_FromPlc} *)
	.TSharpenAxis.NcToPlc AT %IB2110 : NCTOPLC_AXIS_REF;	(*  ~ {LinkedWith:TINC^NC-Task 1 SAF^Axes^Sharpen^Sorties^Sharpen_ToPlc} *)
	.TSharpenEncoder.PlcToNc AT %QB2452 : PLCTONC_AXIS_REF;
	.TSharpenEncoder.NcToPlc AT %IB2528 : NCTOPLC_AXIS_REF;	(*  ~ {LinkedWith:TINC^NC-Task 1 SAF^Axes^SharpenEncoder^Sorties^SharpenEncoder_ToPlc} *)
	.TBarrelAxis.PlcToNc AT %QB2184 : PLCTONC_AXIS_REF;	(*  ~ {LinkedWith:TINC^NC-Task 1 SAF^Axes^Barrel^Entrées^Barrel_FromPlc} *)
	.TBarrelAxis.NcToPlc AT %IB2238 : NCTOPLC_AXIS_REF;	(*  ~ {LinkedWith:TINC^NC-Task 1 SAF^Axes^Barrel^Sorties^Barrel_ToPlc} *)
	.TBrushAxis.PlcToNc AT %QB2312 : PLCTONC_AXIS_REF;	(*  ~ {LinkedWith:TINC^NC-Task 1 SAF^Axes^Brush^Entrées^Brush_FromPlc} *)
	.TBrushAxis.NcToPlc AT %IB2366 : NCTOPLC_AXIS_REF;	(*  ~ {LinkedWith:TINC^NC-Task 1 SAF^Axes^Brush^Sorties^Brush_ToPlc} *)
END_VAR

// ---- Global Variables/Variable_Configuration.TcGVL
{attribute 'Tc2GvlVarNames'}
VAR_CONFIG
END_VAR

// ---- POUs/BG_Serial.TcPOU
PROGRAM BG_Serial
VAR_INPUT
	Enable					: BOOL;
END_VAR
VAR
	bFirstPass				: BOOL	:= TRUE;
	i						: INT;
	(* background communication with the COM port device *)
	as_Control				: ARRAY [1..4] OF SerialLineControlADS;
	as_Config				: ARRAY[1..4] OF ComSerialConfig;
	ab_ControlError			: ARRAY [1..4] OF BOOL;
	an_ControlErrorID			: ARRAY [1..4] OF UDINT;
END_VAR

IF (bFirstPass) THEN
	FOR i:=1 TO C_NB_OF_COM DO
		as_Config[i].ComPort := INT_TO_UDINT(C_COM_NUMBERS[i]);
		IF (as_Config[i].ComPort <> 0) THEN
			as_Config[i].Baudrate :=38400;
			as_Config[i].Parity :=PARITY_NONE;
			as_Config[i].DataBits :=8;
			as_Config[i].StopBits :=STOPBITS_ONE;
			as_Config[i].DTR :=DTR_CTRL_DISABLE;
			as_Config[i].RTS :=RTS_CTRL_DISABLE;
			as_Config[i].CTS :=FALSE;
			as_Config[i].DSR :=FALSE;
		END_IF
	END_FOR
	bFirstPass := FALSE;
END_IF

FOR i:=1 TO C_NB_OF_COM DO
	IF (as_Config[i].ComPort <> 0) THEN
		as_Control[i](
				Connect		:= TRUE,
				SerialCfg		:= as_Config[i],
				TxBuffer		:= TxBuffer_MCR[i],					(* transmit buffer; see global variables *)
				RxBuffer		:= RxBuffer_MCR[i],					(* receive buffer; see global variables *)
				Error		=> ab_ControlError[i],
				ErrorID		=> an_ControlErrorID[i]);
	END_IF
END_FOR

END_PROGRAM

// ---- POUs/MAIN.TcPOU
PROGRAM MAIN
VAR CONSTANT
	iSoftMajorVersion			: INT	:= 2;
	iSoftMinorVersion			: INT	:= 0;

END_VAR
VAR PERSISTENT
	sMachineCnt					: TprodCounter;
	asStickData					: ARRAY[0..1] OF TStickData;
	asStickDataMMI				: ARRAY[0..1] OF TStickDataMMI;
	sStickDataShared			: TStickDataShared;
	sVacuumSettingsMMI			: TVacuumSettingsMMI;
	TAutoSampling				: TAutoSampling;
	bDisableCleanAfterPearling	: BOOL;
	bDisableVision				: BOOL;
	bSpeedModeSlow				: BOOL;
	iMachineWO					: DINT;
	iMachineSN					: INT;
END_VAR
VAR
	sMMI_SyncVar 				: TMachineData;			(* MMI interface data *)
	sMMI_ManualVar 				: TManualData;			(* MMI interface data for manual mode *)
	sMMI_VisionVar				: TVisionData;			(* Vision interface *)
	sMMI_ConfigFileData			: TConfigFileData;
	(* Blocks definitions *)
	TManager					: Manager;
	TLoaderHandler				: LoaderHdl;
	TTableHandler				: TableHdl;
	TPearlingHandler			: PearlingHdl;
	TSharpenHandler				: SharpenHdl;
	TTurnOverHandler			: TurnOverHdl;
	TBarrelHandler				: BarrelHdl;
	TLift1Handler				: LiftHdl;
	TLift2Handler				: LiftHdl;
	TRejectHandler				: RejectHdl;
	TVisionHandler				: VisionHdl;
	TUtilitiesHandler			: UtilitiesHdl;
	eBarrelCmd					: TModuleCommands;
	eLoaderCmd					: TModuleCommands;
	eTableCmd					: TModuleCommands;
	ePearlingCmd				: TModuleCommands;
	eSharpenCmd					: TModuleCommands;
	eTurnOverCmd				: TModuleCommands;
	eLift1Cmd					: TModuleCommands;
	eLift2Cmd					: TModuleCommands;
	eRejectCmd					: TModuleCommands;
	eVisionCmd					: TModuleCommands;
	eUtilitiesCmd				: TModuleCommands;
	TCheckDoors					: TON;
	sGiversTakers				: TStationGiversTakers;
	bFirstCycle					: BOOL				:= TRUE;
	bJobInProgress				: BOOL;
	bPearlingReady4ChangeTool	: BOOL;
	iStickArea2Use				: INT;
	bTableVacuuumNotOk			: BOOL;
	bPearlingHead1IsUsed		: BOOL;
	bPearlingHead2IsUsed		: BOOL;
	eTableSideForLoader			: TTableSide;
	sRunData					: TRunData;
	bTableAspiration13On		: BOOL;
	bTableAspiration24On		: BOOL;
	bLoaderBrushAspirationOn	: BOOL;
	bBrushAspirationOn			: BOOL;
	bSharpenAspirationOn		: BOOL;
	bStopRequest				: BOOL;
	bPauseRequest				: BOOL;
	bLayeringWithTwoParts		: BOOL;
	bNewPlateLift1				: BOOL;
	bNewPlateLift2				: BOOL;
	bNewPlateReject				: BOOL;
	bLoaderVacuumInUse			: BOOL;
	bManInterlockPearling		: BOOL;
	bManInterlockLoader			: BOOL;
	bManInterlockLoaderLift		: BOOL;
	bManInterlockTable			: BOOL;
	bManInterlockTurnOver		: BOOL;
	TJobElapsed					: TIME;
	aiTablePearlsVacuumFlow		: ARRAY[0..1] OF INT;
END_VAR
VAR // added by the converter: edge detectors and wires of the graphical bodies
    _w1, _w3 : TStickData;
    _w2, _w4 : TStickDataMMI;
    _w5 : TStickDataMMIShared;
    _w6 : TVacuumSettingsMMI;
    _w7 : TprodCounter;
    _w8, _w9, _w11, _w12 : INT;
    _w10, _w13, _w14, _w15 : BOOL;
END_VAR

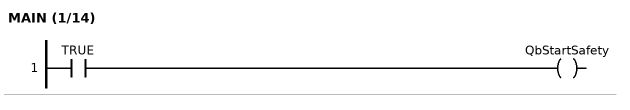
// NETWORK 1
QbStartSafety := TRUE;

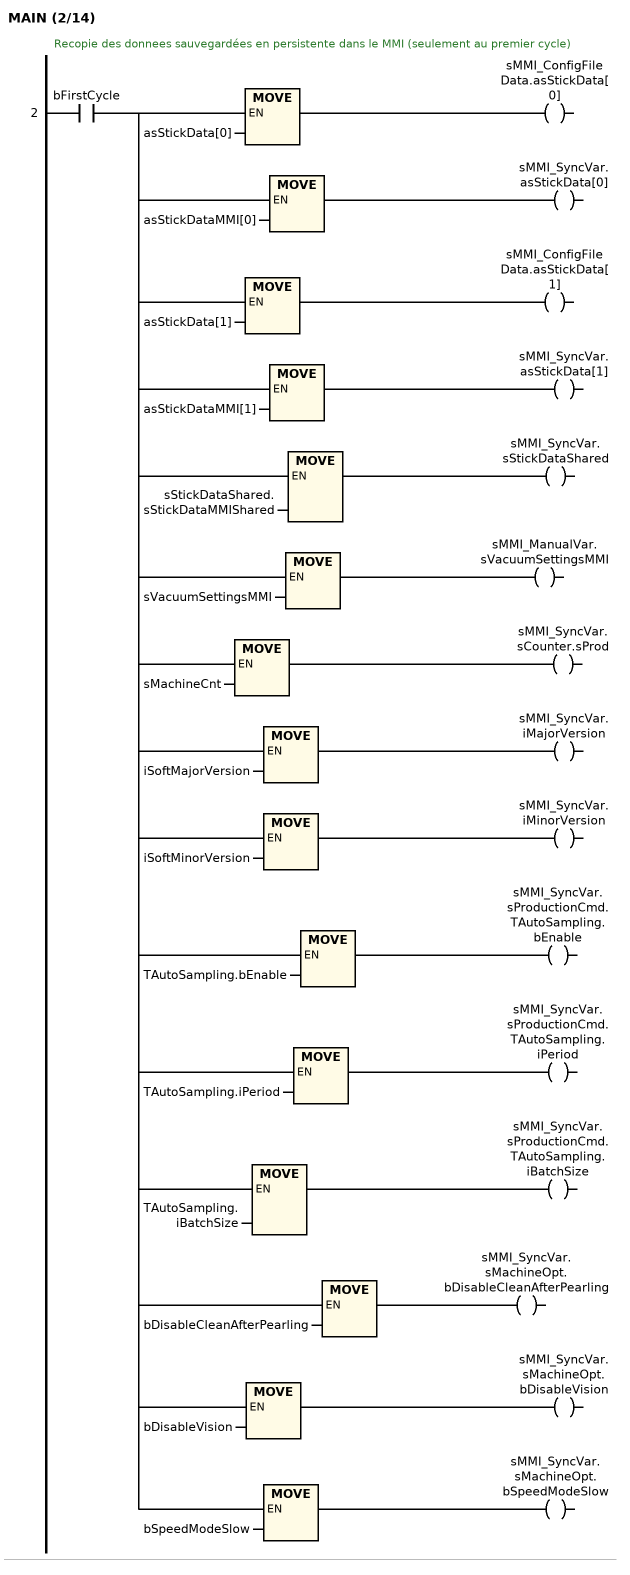
// NETWORK 2
// Recopie des donnees sauvegardées en persistente dans le MMI (seulement au premier cycle)
IF bFirstCycle THEN _w1 := asStickData[0]; END_IF
sMMI_ConfigFileData.asStickData[0] := _w1;
IF bFirstCycle THEN _w2 := asStickDataMMI[0]; END_IF
sMMI_SyncVar.asStickData[0] := _w2;
IF bFirstCycle THEN _w3 := asStickData[1]; END_IF
sMMI_ConfigFileData.asStickData[1] := _w3;
IF bFirstCycle THEN _w4 := asStickDataMMI[1]; END_IF
sMMI_SyncVar.asStickData[1] := _w4;
IF bFirstCycle THEN _w5 := sStickDataShared.sStickDataMMIShared; END_IF
sMMI_SyncVar.sStickDataShared := _w5;
IF bFirstCycle THEN _w6 := sVacuumSettingsMMI; END_IF
sMMI_ManualVar.sVacuumSettingsMMI := _w6;
IF bFirstCycle THEN _w7 := sMachineCnt; END_IF
sMMI_SyncVar.sCounter.sProd := _w7;
IF bFirstCycle THEN _w8 := iSoftMajorVersion; END_IF
sMMI_SyncVar.iMajorVersion := _w8;
IF bFirstCycle THEN _w9 := iSoftMinorVersion; END_IF
sMMI_SyncVar.iMinorVersion := _w9;
IF bFirstCycle THEN _w10 := TAutoSampling.bEnable; END_IF
sMMI_SyncVar.sProductionCmd.TAutoSampling.bEnable := _w10;
IF bFirstCycle THEN _w11 := TAutoSampling.iPeriod; END_IF
sMMI_SyncVar.sProductionCmd.TAutoSampling.iPeriod := _w11;
IF bFirstCycle THEN _w12 := TAutoSampling.iBatchSize; END_IF
sMMI_SyncVar.sProductionCmd.TAutoSampling.iBatchSize := _w12;
IF bFirstCycle THEN _w13 := bDisableCleanAfterPearling; END_IF
sMMI_SyncVar.sMachineOpt.bDisableCleanAfterPearling := _w13;
IF bFirstCycle THEN _w14 := bDisableVision; END_IF
sMMI_SyncVar.sMachineOpt.bDisableVision := _w14;
IF bFirstCycle THEN _w15 := bSpeedModeSlow; END_IF
sMMI_SyncVar.sMachineOpt.bSpeedModeSlow := _w15;

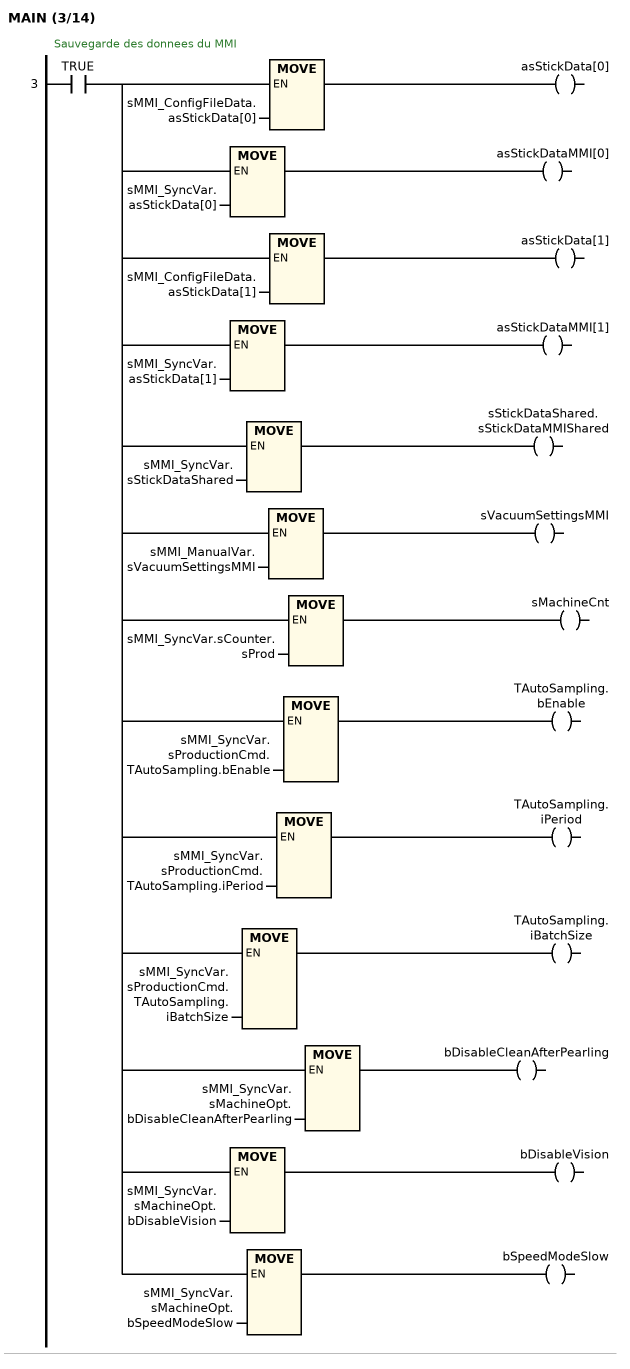
// NETWORK 3
// Sauvegarde des donnees du MMI
asStickData[0] := sMMI_ConfigFileData.asStickData[0];
asStickDataMMI[0] := sMMI_SyncVar.asStickData[0];
asStickData[1] := sMMI_ConfigFileData.asStickData[1];
asStickDataMMI[1] := sMMI_SyncVar.asStickData[1];
sStickDataShared.sStickDataMMIShared := sMMI_SyncVar.sStickDataShared;
sVacuumSettingsMMI := sMMI_ManualVar.sVacuumSettingsMMI;
sMachineCnt := sMMI_SyncVar.sCounter.sProd;
TAutoSampling.bEnable := sMMI_SyncVar.sProductionCmd.TAutoSampling.bEnable;
TAutoSampling.iPeriod := sMMI_SyncVar.sProductionCmd.TAutoSampling.iPeriod;
TAutoSampling.iBatchSize := sMMI_SyncVar.sProductionCmd.TAutoSampling.iBatchSize;
bDisableCleanAfterPearling := sMMI_SyncVar.sMachineOpt.bDisableCleanAfterPearling;
bDisableVision := sMMI_SyncVar.sMachineOpt.bDisableVision;
bSpeedModeSlow := sMMI_SyncVar.sMachineOpt.bSpeedModeSlow;

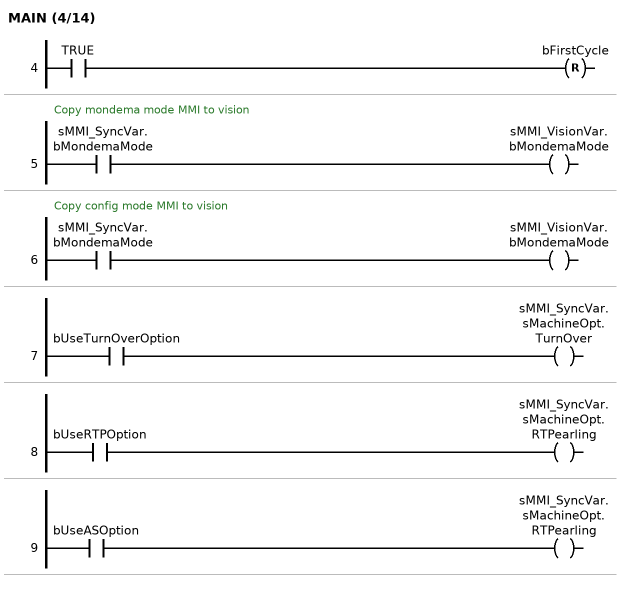
// NETWORK 4
bFirstCycle R= TRUE;

// NETWORK 5
// Copy mondema mode MMI to vision
sMMI_VisionVar.bMondemaMode := sMMI_SyncVar.bMondemaMode;

// NETWORK 6
// Copy config mode MMI to vision
sMMI_VisionVar.bMondemaMode := sMMI_SyncVar.bMondemaMode;

// NETWORK 7
sMMI_SyncVar.sMachineOpt.TurnOver := bUseTurnOverOption;

// NETWORK 8
sMMI_SyncVar.sMachineOpt.RTPearling := bUseRTPOption;

// NETWORK 9
sMMI_SyncVar.sMachineOpt.RTPearling := bUseASOption;

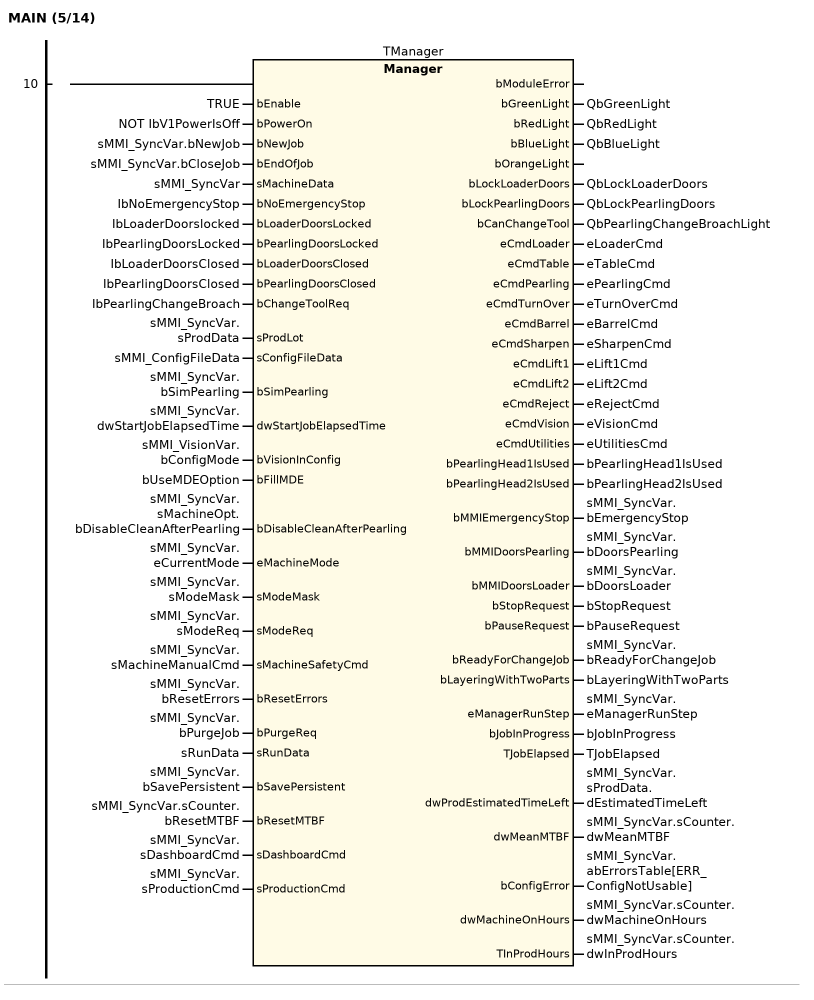
// NETWORK 10
TManager(
    bEnable := TRUE,
    bPowerOn := NOT IbV1PowerIsOff,
    bNewJob := sMMI_SyncVar.bNewJob,
    bEndOfJob := sMMI_SyncVar.bCloseJob,
    sMachineData := sMMI_SyncVar,
    bNoEmergencyStop := IbNoEmergencyStop,
    bLoaderDoorsLocked := IbLoaderDoorslocked,
    bPearlingDoorsLocked := IbPearlingDoorsLocked,
    bLoaderDoorsClosed := IbLoaderDoorsClosed,
    bPearlingDoorsClosed := IbPearlingDoorsClosed,
    bChangeToolReq := IbPearlingChangeBroach,
    sProdLot := sMMI_SyncVar.sProdData,
    sConfigFileData := sMMI_ConfigFileData,
    bSimPearling := sMMI_SyncVar.bSimPearling,
    dwStartJobElapsedTime := sMMI_SyncVar.dwStartJobElapsedTime,
    bVisionInConfig := sMMI_VisionVar.bConfigMode,
    bFillMDE := bUseMDEOption,
    bDisableCleanAfterPearling := sMMI_SyncVar.sMachineOpt.bDisableCleanAfterPearling,
    eMachineMode := sMMI_SyncVar.eCurrentMode,
    sModeMask := sMMI_SyncVar.sModeMask,
    sModeReq := sMMI_SyncVar.sModeReq,
    sMachineSafetyCmd := sMMI_SyncVar.sMachineManualCmd,
    bResetErrors := sMMI_SyncVar.bResetErrors,
    bPurgeReq := sMMI_SyncVar.bPurgeJob,
    sRunData := sRunData,
    bSavePersistent := sMMI_SyncVar.bSavePersistent,
    bResetMTBF := sMMI_SyncVar.sCounter.bResetMTBF,
    sDashboardCmd := sMMI_SyncVar.sDashboardCmd,
    sProductionCmd := sMMI_SyncVar.sProductionCmd,
    bGreenLight => QbGreenLight,
    bRedLight => QbRedLight,
    bBlueLight => QbBlueLight,
    bLockLoaderDoors => QbLockLoaderDoors,
    bLockPearlingDoors => QbLockPearlingDoors,
    bCanChangeTool => QbPearlingChangeBroachLight,
    eCmdLoader => eLoaderCmd,
    eCmdTable => eTableCmd,
    eCmdPearling => ePearlingCmd,
    eCmdTurnOver => eTurnOverCmd,
    eCmdBarrel => eBarrelCmd,
    eCmdSharpen => eSharpenCmd,
    eCmdLift1 => eLift1Cmd,
    eCmdLift2 => eLift2Cmd,
    eCmdReject => eRejectCmd,
    eCmdVision => eVisionCmd,
    eCmdUtilities => eUtilitiesCmd,
    bPearlingHead1IsUsed => bPearlingHead1IsUsed,
    bPearlingHead2IsUsed => bPearlingHead2IsUsed,
    bMMIEmergencyStop => sMMI_SyncVar.bEmergencyStop,
    bMMIDoorsPearling => sMMI_SyncVar.bDoorsPearling,
    bMMIDoorsLoader => sMMI_SyncVar.bDoorsLoader,
    bStopRequest => bStopRequest,
    bPauseRequest => bPauseRequest,
    bReadyForChangeJob => sMMI_SyncVar.bReadyForChangeJob,
    bLayeringWithTwoParts => bLayeringWithTwoParts,
    eManagerRunStep => sMMI_SyncVar.eManagerRunStep,
    bJobInProgress => bJobInProgress,
    TJobElapsed => TJobElapsed,
    dwProdEstimatedTimeLeft => sMMI_SyncVar.sProdData.dEstimatedTimeLeft,
    dwMeanMTBF => sMMI_SyncVar.sCounter.dwMeanMTBF,
    bConfigError => sMMI_SyncVar.abErrorsTable[ERR_ConfigNotUsable],
    dwMachineOnHours => sMMI_SyncVar.sCounter.dwMachineOnHours,
    TInProdHours => sMMI_SyncVar.sCounter.dwInProdHours); // Manager

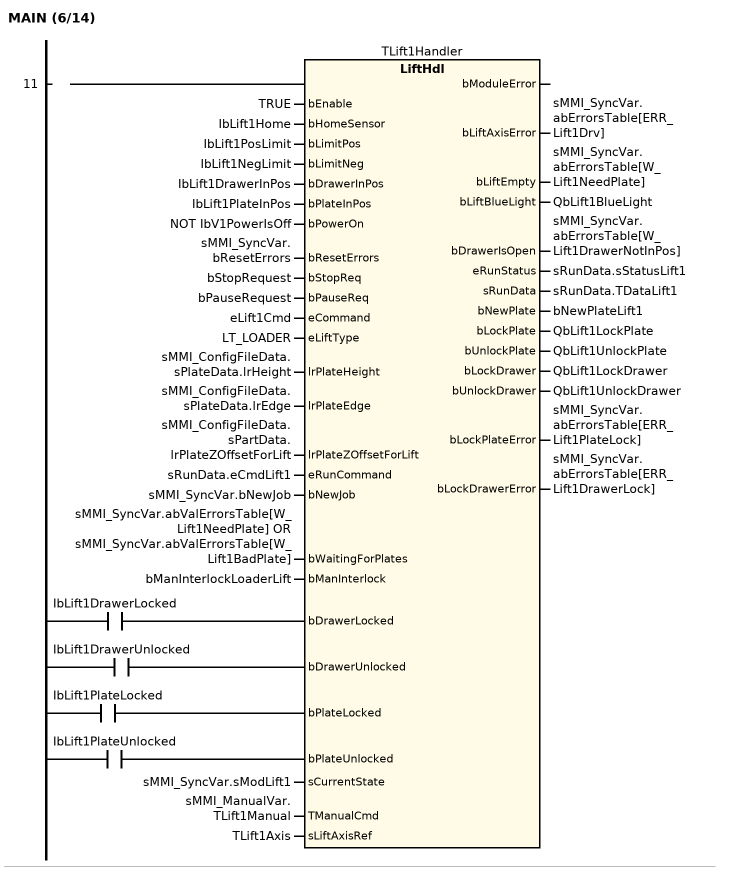
// NETWORK 11
TLift1Handler(
    bEnable := TRUE,
    bHomeSensor := IbLift1Home,
    bLimitPos := IbLift1PosLimit,
    bLimitNeg := IbLift1NegLimit,
    bDrawerInPos := IbLift1DrawerInPos,
    bPlateInPos := IbLift1PlateInPos,
    bPowerOn := NOT IbV1PowerIsOff,
    bResetErrors := sMMI_SyncVar.bResetErrors,
    bStopReq := bStopRequest,
    bPauseReq := bPauseRequest,
    eCommand := eLift1Cmd,
    eLiftType := LT_LOADER,
    lrPlateHeight := sMMI_ConfigFileData.sPlateData.lrHeight,
    lrPlateEdge := sMMI_ConfigFileData.sPlateData.lrEdge,
    lrPlateZOffsetForLift := sMMI_ConfigFileData.sPartData.lrPlateZOffsetForLift,
    eRunCommand := sRunData.eCmdLift1,
    bNewJob := sMMI_SyncVar.bNewJob,
    bWaitingForPlates := sMMI_SyncVar.abValErrorsTable[W_Lift1NeedPlate] OR sMMI_SyncVar.abValErrorsTable[W_Lift1BadPlate],
    bManInterlock := bManInterlockLoaderLift,
    bDrawerLocked := IbLift1DrawerLocked,
    bDrawerUnlocked := IbLift1DrawerUnlocked,
    bPlateLocked := IbLift1PlateLocked,
    bPlateUnlocked := IbLift1PlateUnlocked,
    sCurrentState := sMMI_SyncVar.sModLift1,
    TManualCmd := sMMI_ManualVar.TLift1Manual,
    sLiftAxisRef := TLift1Axis,
    bLiftAxisError => sMMI_SyncVar.abErrorsTable[ERR_Lift1Drv],
    bLiftEmpty => sMMI_SyncVar.abErrorsTable[W_Lift1NeedPlate],
    bLiftBlueLight => QbLift1BlueLight,
    bDrawerIsOpen => sMMI_SyncVar.abErrorsTable[W_Lift1DrawerNotInPos],
    eRunStatus => sRunData.sStatusLift1,
    sRunData => sRunData.TDataLift1,
    bNewPlate => bNewPlateLift1,
    bLockPlate => QbLift1LockPlate,
    bUnlockPlate => QbLift1UnlockPlate,
    bLockDrawer => QbLift1LockDrawer,
    bUnlockDrawer => QbLift1UnlockDrawer,
    bLockPlateError => sMMI_SyncVar.abErrorsTable[ERR_Lift1PlateLock],
    bLockDrawerError => sMMI_SyncVar.abErrorsTable[ERR_Lift1DrawerLock]); // LiftHdl

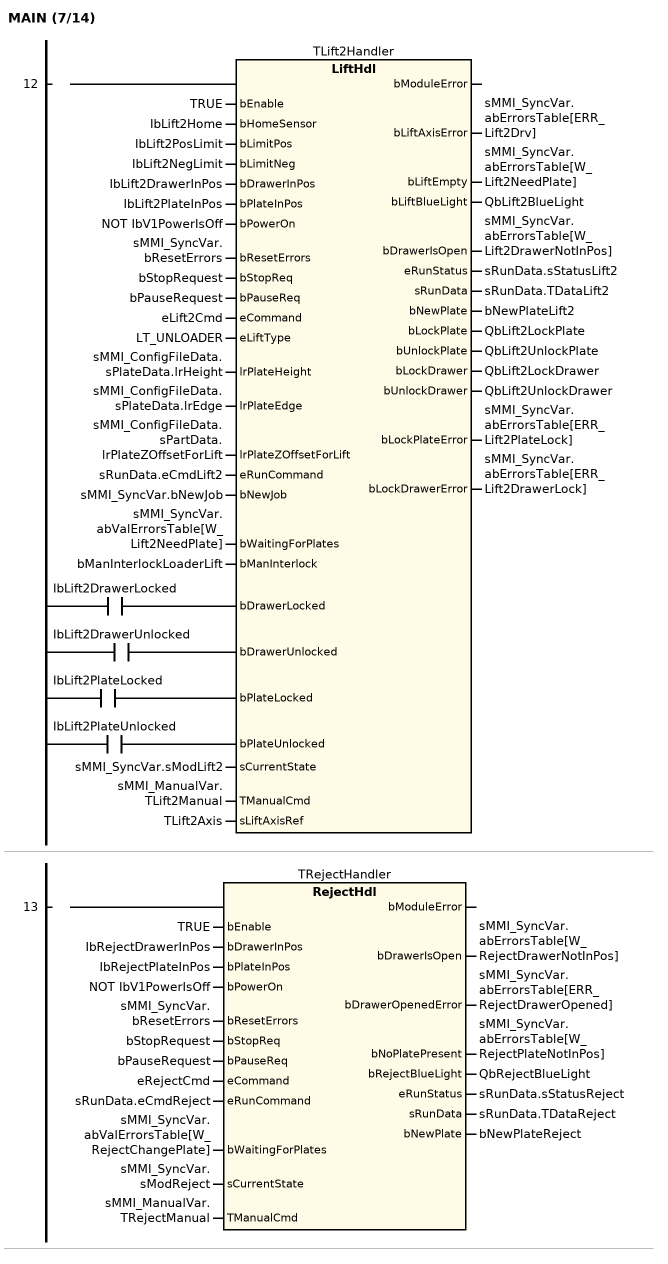
// NETWORK 12
TLift2Handler(
    bEnable := TRUE,
    bHomeSensor := IbLift2Home,
    bLimitPos := IbLift2PosLimit,
    bLimitNeg := IbLift2NegLimit,
    bDrawerInPos := IbLift2DrawerInPos,
    bPlateInPos := IbLift2PlateInPos,
    bPowerOn := NOT IbV1PowerIsOff,
    bResetErrors := sMMI_SyncVar.bResetErrors,
    bStopReq := bStopRequest,
    bPauseReq := bPauseRequest,
    eCommand := eLift2Cmd,
    eLiftType := LT_UNLOADER,
    lrPlateHeight := sMMI_ConfigFileData.sPlateData.lrHeight,
    lrPlateEdge := sMMI_ConfigFileData.sPlateData.lrEdge,
    lrPlateZOffsetForLift := sMMI_ConfigFileData.sPartData.lrPlateZOffsetForLift,
    eRunCommand := sRunData.eCmdLift2,
    bNewJob := sMMI_SyncVar.bNewJob,
    bWaitingForPlates := sMMI_SyncVar.abValErrorsTable[W_Lift2NeedPlate],
    bManInterlock := bManInterlockLoaderLift,
    bDrawerLocked := IbLift2DrawerLocked,
    bDrawerUnlocked := IbLift2DrawerUnlocked,
    bPlateLocked := IbLift2PlateLocked,
    bPlateUnlocked := IbLift2PlateUnlocked,
    sCurrentState := sMMI_SyncVar.sModLift2,
    TManualCmd := sMMI_ManualVar.TLift2Manual,
    sLiftAxisRef := TLift2Axis,
    bLiftAxisError => sMMI_SyncVar.abErrorsTable[ERR_Lift2Drv],
    bLiftEmpty => sMMI_SyncVar.abErrorsTable[W_Lift2NeedPlate],
    bLiftBlueLight => QbLift2BlueLight,
    bDrawerIsOpen => sMMI_SyncVar.abErrorsTable[W_Lift2DrawerNotInPos],
    eRunStatus => sRunData.sStatusLift2,
    sRunData => sRunData.TDataLift2,
    bNewPlate => bNewPlateLift2,
    bLockPlate => QbLift2LockPlate,
    bUnlockPlate => QbLift2UnlockPlate,
    bLockDrawer => QbLift2LockDrawer,
    bUnlockDrawer => QbLift2UnlockDrawer,
    bLockPlateError => sMMI_SyncVar.abErrorsTable[ERR_Lift2PlateLock],
    bLockDrawerError => sMMI_SyncVar.abErrorsTable[ERR_Lift2DrawerLock]); // LiftHdl

// NETWORK 13
TRejectHandler(
    bEnable := TRUE,
    bDrawerInPos := IbRejectDrawerInPos,
    bPlateInPos := IbRejectPlateInPos,
    bPowerOn := NOT IbV1PowerIsOff,
    bResetErrors := sMMI_SyncVar.bResetErrors,
    bStopReq := bStopRequest,
    bPauseReq := bPauseRequest,
    eCommand := eRejectCmd,
    eRunCommand := sRunData.eCmdReject,
    bWaitingForPlates := sMMI_SyncVar.abValErrorsTable[W_RejectChangePlate],
    sCurrentState := sMMI_SyncVar.sModReject,
    TManualCmd := sMMI_ManualVar.TRejectManual,
    bDrawerIsOpen => sMMI_SyncVar.abErrorsTable[W_RejectDrawerNotInPos],
    bDrawerOpenedError => sMMI_SyncVar.abErrorsTable[ERR_RejectDrawerOpened],
    bNoPlatePresent => sMMI_SyncVar.abErrorsTable[W_RejectPlateNotInPos],
    bRejectBlueLight => QbRejectBlueLight,
    eRunStatus => sRunData.sStatusReject,
    sRunData => sRunData.TDataReject,
    bNewPlate => bNewPlateReject); // RejectHdl

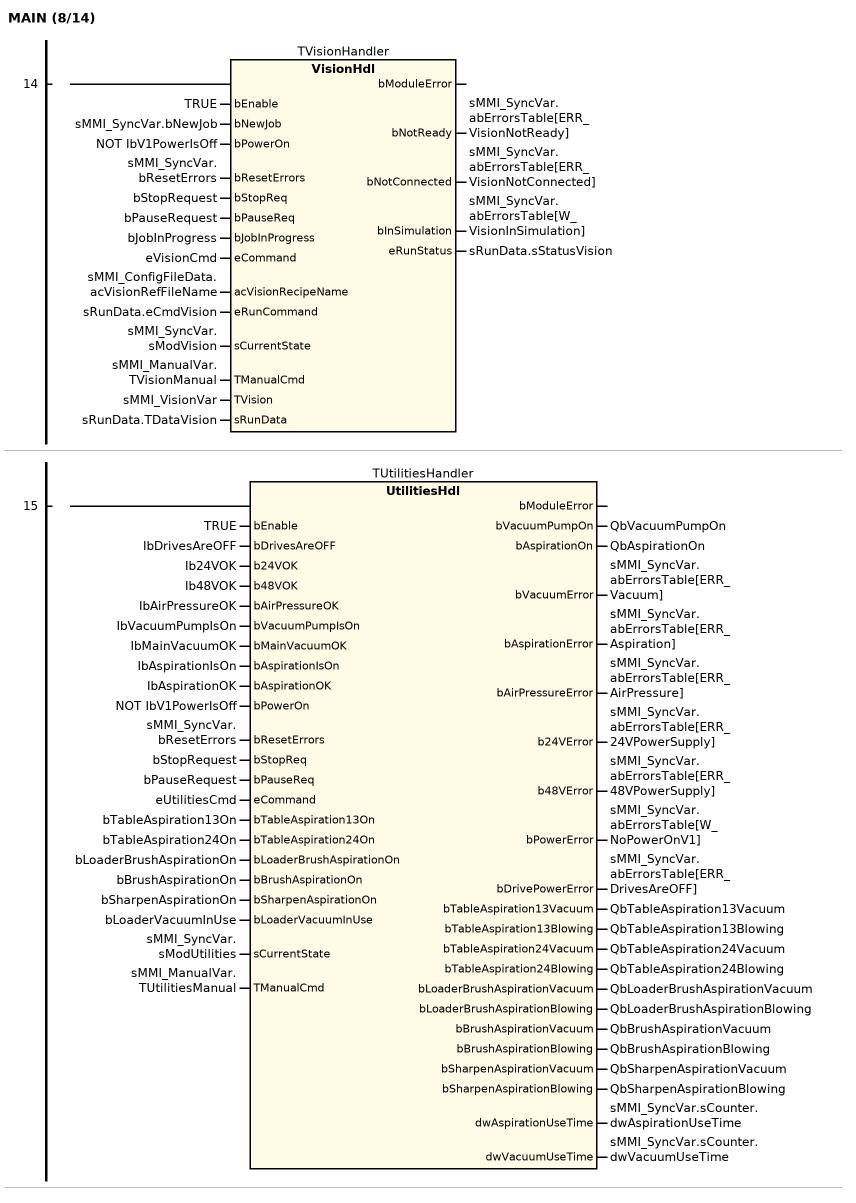
// NETWORK 14
TVisionHandler(
    bEnable := TRUE,
    bNewJob := sMMI_SyncVar.bNewJob,
    bPowerOn := NOT IbV1PowerIsOff,
    bResetErrors := sMMI_SyncVar.bResetErrors,
    bStopReq := bStopRequest,
    bPauseReq := bPauseRequest,
    bJobInProgress := bJobInProgress,
    eCommand := eVisionCmd,
    acVisionRecipeName := sMMI_ConfigFileData.acVisionRefFileName,
    eRunCommand := sRunData.eCmdVision,
    sCurrentState := sMMI_SyncVar.sModVision,
    TManualCmd := sMMI_ManualVar.TVisionManual,
    TVision := sMMI_VisionVar,
    sRunData := sRunData.TDataVision,
    bNotReady => sMMI_SyncVar.abErrorsTable[ERR_VisionNotReady],
    bNotConnected => sMMI_SyncVar.abErrorsTable[ERR_VisionNotConnected],
    bInSimulation => sMMI_SyncVar.abErrorsTable[W_VisionInSimulation],
    eRunStatus => sRunData.sStatusVision); // VisionHdl

// NETWORK 15
TUtilitiesHandler(
    bEnable := TRUE,
    bDrivesAreOFF := IbDrivesAreOFF,
    b24VOK := Ib24VOK,
    b48VOK := Ib48VOK,
    bAirPressureOK := IbAirPressureOK,
    bVacuumPumpIsOn := IbVacuumPumpIsOn,
    bMainVacuumOK := IbMainVacuumOK,
    bAspirationIsOn := IbAspirationIsOn,
    bAspirationOK := IbAspirationOK,
    bPowerOn := NOT IbV1PowerIsOff,
    bResetErrors := sMMI_SyncVar.bResetErrors,
    bStopReq := bStopRequest,
    bPauseReq := bPauseRequest,
    eCommand := eUtilitiesCmd,
    bTableAspiration13On := bTableAspiration13On,
    bTableAspiration24On := bTableAspiration24On,
    bLoaderBrushAspirationOn := bLoaderBrushAspirationOn,
    bBrushAspirationOn := bBrushAspirationOn,
    bSharpenAspirationOn := bSharpenAspirationOn,
    bLoaderVacuumInUse := bLoaderVacuumInUse,
    sCurrentState := sMMI_SyncVar.sModUtilities,
    TManualCmd := sMMI_ManualVar.TUtilitiesManual,
    bVacuumPumpOn => QbVacuumPumpOn,
    bAspirationOn => QbAspirationOn,
    bVacuumError => sMMI_SyncVar.abErrorsTable[ERR_Vacuum],
    bAspirationError => sMMI_SyncVar.abErrorsTable[ERR_Aspiration],
    bAirPressureError => sMMI_SyncVar.abErrorsTable[ERR_AirPressure],
    b24VError => sMMI_SyncVar.abErrorsTable[ERR_24VPowerSupply],
    b48VError => sMMI_SyncVar.abErrorsTable[ERR_48VPowerSupply],
    bPowerError => sMMI_SyncVar.abErrorsTable[W_NoPowerOnV1],
    bDrivePowerError => sMMI_SyncVar.abErrorsTable[ERR_DrivesAreOFF],
    bTableAspiration13Vacuum => QbTableAspiration13Vacuum,
    bTableAspiration13Blowing => QbTableAspiration13Blowing,
    bTableAspiration24Vacuum => QbTableAspiration24Vacuum,
    bTableAspiration24Blowing => QbTableAspiration24Blowing,
    bLoaderBrushAspirationVacuum => QbLoaderBrushAspirationVacuum,
    bLoaderBrushAspirationBlowing => QbLoaderBrushAspirationBlowing,
    bBrushAspirationVacuum => QbBrushAspirationVacuum,
    bBrushAspirationBlowing => QbBrushAspirationBlowing,
    bSharpenAspirationVacuum => QbSharpenAspirationVacuum,
    bSharpenAspirationBlowing => QbSharpenAspirationBlowing,
    dwAspirationUseTime => sMMI_SyncVar.sCounter.dwAspirationUseTime,
    dwVacuumUseTime => sMMI_SyncVar.sCounter.dwVacuumUseTime); // UtilitiesHdl

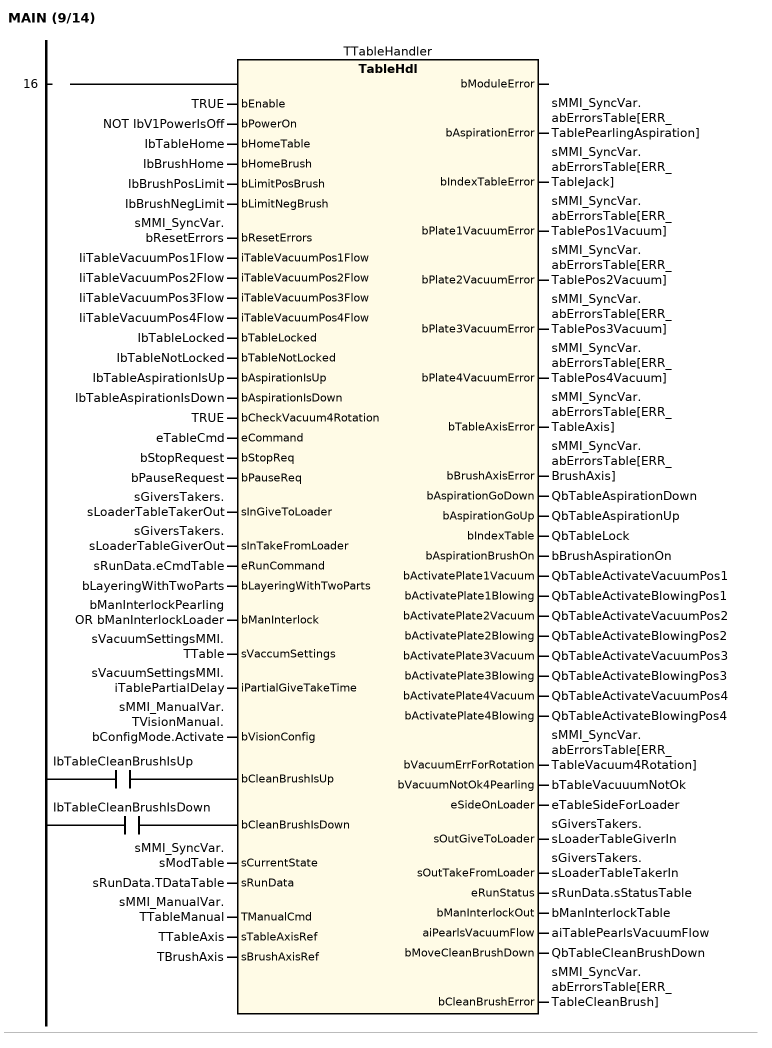
// NETWORK 16
TTableHandler(
    bEnable := TRUE,
    bPowerOn := NOT IbV1PowerIsOff,
    bHomeTable := IbTableHome,
    bHomeBrush := IbBrushHome,
    bLimitPosBrush := IbBrushPosLimit,
    bLimitNegBrush := IbBrushNegLimit,
    bResetErrors := sMMI_SyncVar.bResetErrors,
    iTableVacuumPos1Flow := IiTableVacuumPos1Flow,
    iTableVacuumPos2Flow := IiTableVacuumPos2Flow,
    iTableVacuumPos3Flow := IiTableVacuumPos3Flow,
    iTableVacuumPos4Flow := IiTableVacuumPos4Flow,
    bTableLocked := IbTableLocked,
    bTableNotLocked := IbTableNotLocked,
    bAspirationIsUp := IbTableAspirationIsUp,
    bAspirationIsDown := IbTableAspirationIsDown,
    bCheckVacuum4Rotation := TRUE,
    eCommand := eTableCmd,
    bStopReq := bStopRequest,
    bPauseReq := bPauseRequest,
    sInGiveToLoader := sGiversTakers.sLoaderTableTakerOut,
    sInTakeFromLoader := sGiversTakers.sLoaderTableGiverOut,
    eRunCommand := sRunData.eCmdTable,
    bLayeringWithTwoParts := bLayeringWithTwoParts,
    bManInterlock := bManInterlockPearling OR bManInterlockLoader,
    sVaccumSettings := sVacuumSettingsMMI.TTable,
    iPartialGiveTakeTime := sVacuumSettingsMMI.iTablePartialDelay,
    bVisionConfig := sMMI_ManualVar.TVisionManual.bConfigMode.Activate,
    bCleanBrushIsUp := IbTableCleanBrushIsUp,
    bCleanBrushIsDown := IbTableCleanBrushIsDown,
    sCurrentState := sMMI_SyncVar.sModTable,
    sRunData := sRunData.TDataTable,
    TManualCmd := sMMI_ManualVar.TTableManual,
    sTableAxisRef := TTableAxis,
    sBrushAxisRef := TBrushAxis,
    bAspirationError => sMMI_SyncVar.abErrorsTable[ERR_TablePearlingAspiration],
    bIndexTableError => sMMI_SyncVar.abErrorsTable[ERR_TableJack],
    bPlate1VacuumError => sMMI_SyncVar.abErrorsTable[ERR_TablePos1Vacuum],
    bPlate2VacuumError => sMMI_SyncVar.abErrorsTable[ERR_TablePos2Vacuum],
    bPlate3VacuumError => sMMI_SyncVar.abErrorsTable[ERR_TablePos3Vacuum],
    bPlate4VacuumError => sMMI_SyncVar.abErrorsTable[ERR_TablePos4Vacuum],
    bTableAxisError => sMMI_SyncVar.abErrorsTable[ERR_TableAxis],
    bBrushAxisError => sMMI_SyncVar.abErrorsTable[ERR_BrushAxis],
    bAspirationGoDown => QbTableAspirationDown,
    bAspirationGoUp => QbTableAspirationUp,
    bIndexTable => QbTableLock,
    bAspirationBrushOn => bBrushAspirationOn,
    bActivatePlate1Vacuum => QbTableActivateVacuumPos1,
    bActivatePlate1Blowing => QbTableActivateBlowingPos1,
    bActivatePlate2Vacuum => QbTableActivateVacuumPos2,
    bActivatePlate2Blowing => QbTableActivateBlowingPos2,
    bActivatePlate3Vacuum => QbTableActivateVacuumPos3,
    bActivatePlate3Blowing => QbTableActivateBlowingPos3,
    bActivatePlate4Vacuum => QbTableActivateVacuumPos4,
    bActivatePlate4Blowing => QbTableActivateBlowingPos4,
    bVacuumErrForRotation => sMMI_SyncVar.abErrorsTable[ERR_TableVacuum4Rotation],
    bVacuumNotOk4Pearling => bTableVacuuumNotOk,
    eSideOnLoader => eTableSideForLoader,
    sOutGiveToLoader => sGiversTakers.sLoaderTableGiverIn,
    sOutTakeFromLoader => sGiversTakers.sLoaderTableTakerIn,
    eRunStatus => sRunData.sStatusTable,
    bManInterlockOut => bManInterlockTable,
    aiPearlsVacuumFlow => aiTablePearlsVacuumFlow,
    bMoveCleanBrushDown => QbTableCleanBrushDown,
    bCleanBrushError => sMMI_SyncVar.abErrorsTable[ERR_TableCleanBrush]); // TableHdl

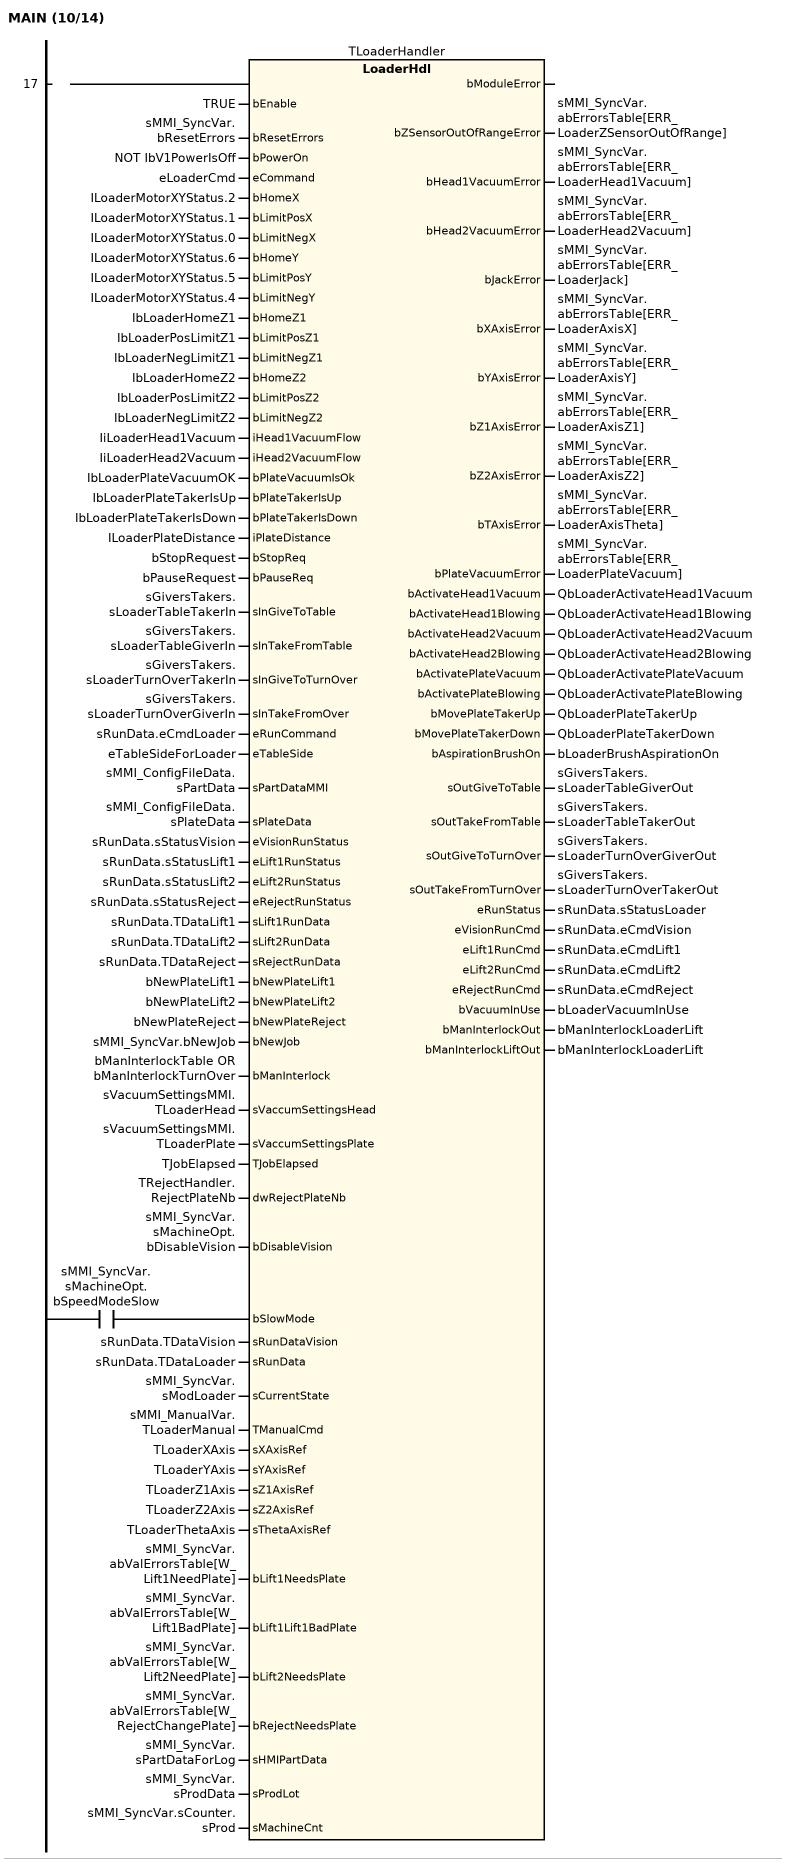
// NETWORK 17
TLoaderHandler(
    bEnable := TRUE,
    bResetErrors := sMMI_SyncVar.bResetErrors,
    bPowerOn := NOT IbV1PowerIsOff,
    eCommand := eLoaderCmd,
    bHomeX := ILoaderMotorXYStatus.2,
    bLimitPosX := ILoaderMotorXYStatus.1,
    bLimitNegX := ILoaderMotorXYStatus.0,
    bHomeY := ILoaderMotorXYStatus.6,
    bLimitPosY := ILoaderMotorXYStatus.5,
    bLimitNegY := ILoaderMotorXYStatus.4,
    bHomeZ1 := IbLoaderHomeZ1,
    bLimitPosZ1 := IbLoaderPosLimitZ1,
    bLimitNegZ1 := IbLoaderNegLimitZ1,
    bHomeZ2 := IbLoaderHomeZ2,
    bLimitPosZ2 := IbLoaderPosLimitZ2,
    bLimitNegZ2 := IbLoaderNegLimitZ2,
    iHead1VacuumFlow := IiLoaderHead1Vacuum,
    iHead2VacuumFlow := IiLoaderHead2Vacuum,
    bPlateVacuumIsOk := IbLoaderPlateVacuumOK,
    bPlateTakerIsUp := IbLoaderPlateTakerIsUp,
    bPlateTakerIsDown := IbLoaderPlateTakerIsDown,
    iPlateDistance := ILoaderPlateDistance,
    bStopReq := bStopRequest,
    bPauseReq := bPauseRequest,
    sInGiveToTable := sGiversTakers.sLoaderTableTakerIn,
    sInTakeFromTable := sGiversTakers.sLoaderTableGiverIn,
    sInGiveToTurnOver := sGiversTakers.sLoaderTurnOverTakerIn,
    sInTakeFromOver := sGiversTakers.sLoaderTurnOverGiverIn,
    eRunCommand := sRunData.eCmdLoader,
    eTableSide := eTableSideForLoader,
    sPartDataMMI := sMMI_ConfigFileData.sPartData,
    sPlateData := sMMI_ConfigFileData.sPlateData,
    eVisionRunStatus := sRunData.sStatusVision,
    eLift1RunStatus := sRunData.sStatusLift1,
    eLift2RunStatus := sRunData.sStatusLift2,
    eRejectRunStatus := sRunData.sStatusReject,
    sLift1RunData := sRunData.TDataLift1,
    sLift2RunData := sRunData.TDataLift2,
    sRejectRunData := sRunData.TDataReject,
    bNewPlateLift1 := bNewPlateLift1,
    bNewPlateLift2 := bNewPlateLift2,
    bNewPlateReject := bNewPlateReject,
    bNewJob := sMMI_SyncVar.bNewJob,
    bManInterlock := bManInterlockTable OR bManInterlockTurnOver,
    sVaccumSettingsHead := sVacuumSettingsMMI.TLoaderHead,
    sVaccumSettingsPlate := sVacuumSettingsMMI.TLoaderPlate,
    TJobElapsed := TJobElapsed,
    dwRejectPlateNb := TRejectHandler.RejectPlateNb,
    bDisableVision := sMMI_SyncVar.sMachineOpt.bDisableVision,
    bSlowMode := sMMI_SyncVar.sMachineOpt.bSpeedModeSlow,
    sRunDataVision := sRunData.TDataVision,
    sRunData := sRunData.TDataLoader,
    sCurrentState := sMMI_SyncVar.sModLoader,
    TManualCmd := sMMI_ManualVar.TLoaderManual,
    sXAxisRef := TLoaderXAxis,
    sYAxisRef := TLoaderYAxis,
    sZ1AxisRef := TLoaderZ1Axis,
    sZ2AxisRef := TLoaderZ2Axis,
    sThetaAxisRef := TLoaderThetaAxis,
    bLift1NeedsPlate := sMMI_SyncVar.abValErrorsTable[W_Lift1NeedPlate],
    bLift1Lift1BadPlate := sMMI_SyncVar.abValErrorsTable[W_Lift1BadPlate],
    bLift2NeedsPlate := sMMI_SyncVar.abValErrorsTable[W_Lift2NeedPlate],
    bRejectNeedsPlate := sMMI_SyncVar.abValErrorsTable[W_RejectChangePlate],
    sHMIPartData := sMMI_SyncVar.sPartDataForLog,
    sProdLot := sMMI_SyncVar.sProdData,
    sMachineCnt := sMMI_SyncVar.sCounter.sProd,
    bZSensorOutOfRangeError => sMMI_SyncVar.abErrorsTable[ERR_LoaderZSensorOutOfRange],
    bHead1VacuumError => sMMI_SyncVar.abErrorsTable[ERR_LoaderHead1Vacuum],
    bHead2VacuumError => sMMI_SyncVar.abErrorsTable[ERR_LoaderHead2Vacuum],
    bJackError => sMMI_SyncVar.abErrorsTable[ERR_LoaderJack],
    bXAxisError => sMMI_SyncVar.abErrorsTable[ERR_LoaderAxisX],
    bYAxisError => sMMI_SyncVar.abErrorsTable[ERR_LoaderAxisY],
    bZ1AxisError => sMMI_SyncVar.abErrorsTable[ERR_LoaderAxisZ1],
    bZ2AxisError => sMMI_SyncVar.abErrorsTable[ERR_LoaderAxisZ2],
    bTAxisError => sMMI_SyncVar.abErrorsTable[ERR_LoaderAxisTheta],
    bPlateVacuumError => sMMI_SyncVar.abErrorsTable[ERR_LoaderPlateVacuum],
    bActivateHead1Vacuum => QbLoaderActivateHead1Vacuum,
    bActivateHead1Blowing => QbLoaderActivateHead1Blowing,
    bActivateHead2Vacuum => QbLoaderActivateHead2Vacuum,
    bActivateHead2Blowing => QbLoaderActivateHead2Blowing,
    bActivatePlateVacuum => QbLoaderActivatePlateVacuum,
    bActivatePlateBlowing => QbLoaderActivatePlateBlowing,
    bMovePlateTakerUp => QbLoaderPlateTakerUp,
    bMovePlateTakerDown => QbLoaderPlateTakerDown,
    bAspirationBrushOn => bLoaderBrushAspirationOn,
    sOutGiveToTable => sGiversTakers.sLoaderTableGiverOut,
    sOutTakeFromTable => sGiversTakers.sLoaderTableTakerOut,
    sOutGiveToTurnOver => sGiversTakers.sLoaderTurnOverGiverOut,
    sOutTakeFromTurnOver => sGiversTakers.sLoaderTurnOverTakerOut,
    eRunStatus => sRunData.sStatusLoader,
    eVisionRunCmd => sRunData.eCmdVision,
    eLift1RunCmd => sRunData.eCmdLift1,
    eLift2RunCmd => sRunData.eCmdLift2,
    eRejectRunCmd => sRunData.eCmdReject,
    bVacuumInUse => bLoaderVacuumInUse,
    bManInterlockOut => bManInterlockLoaderLift,
    bManInterlockLiftOut => bManInterlockLoaderLift); // LoaderHdl

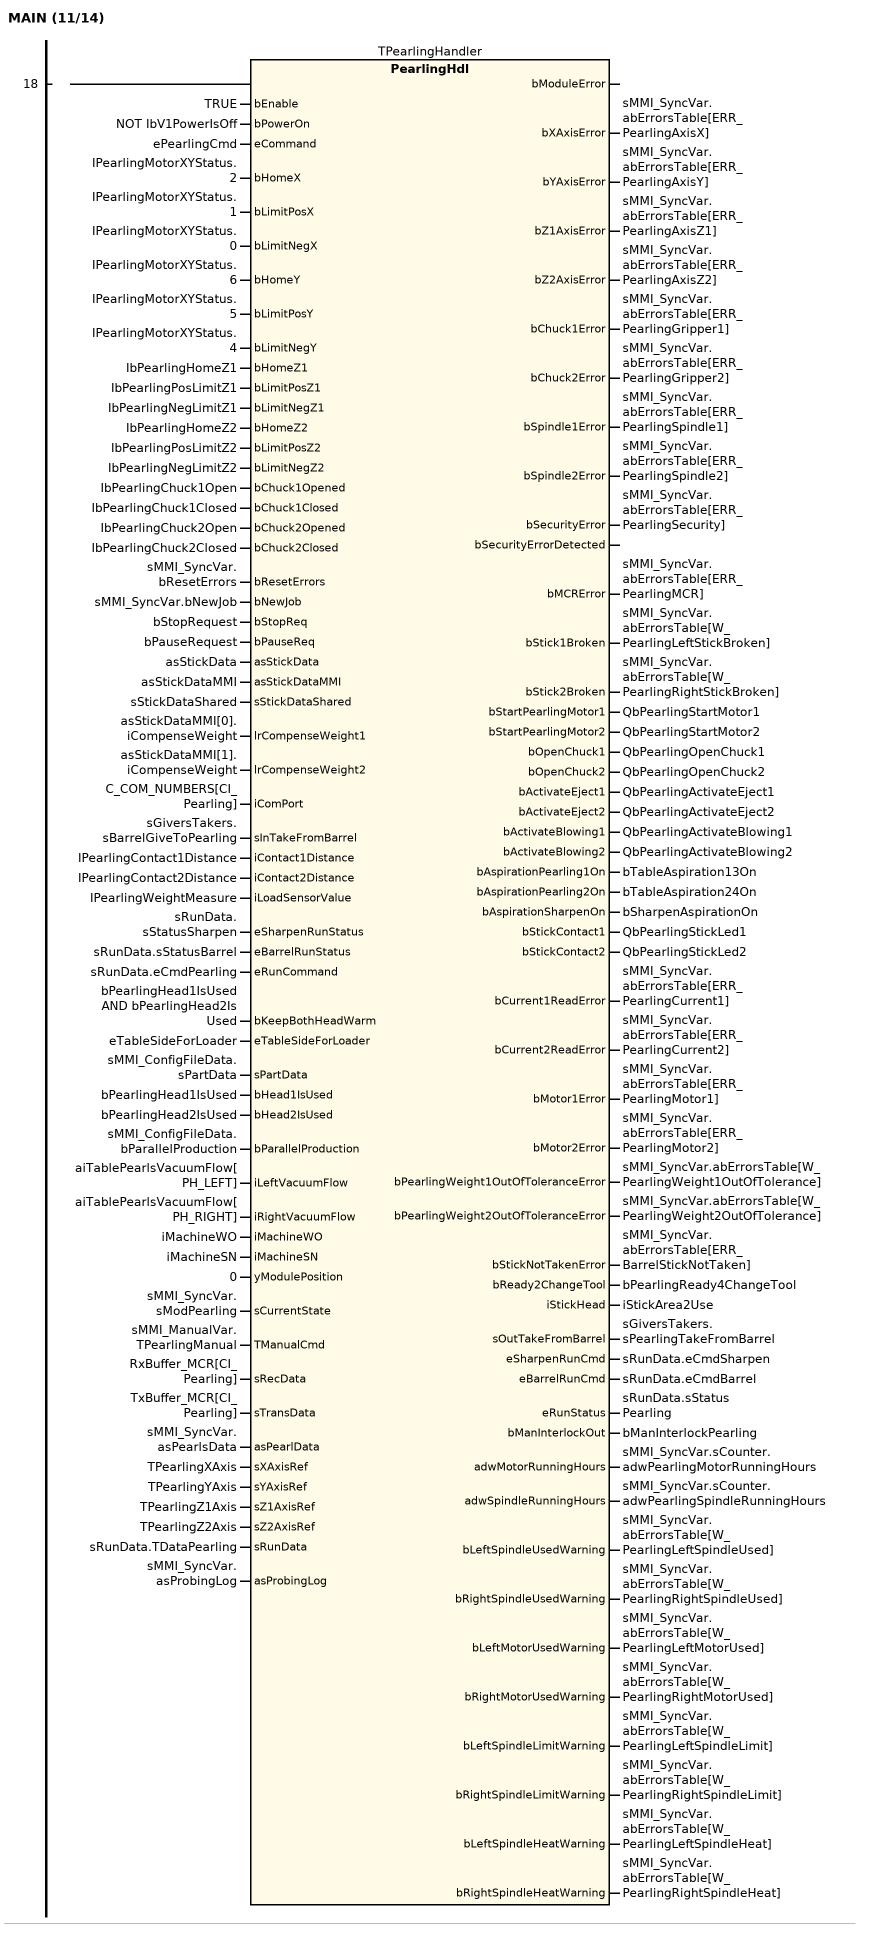
// NETWORK 18
TPearlingHandler(
    bEnable := TRUE,
    bPowerOn := NOT IbV1PowerIsOff,
    eCommand := ePearlingCmd,
    bHomeX := IPearlingMotorXYStatus.2,
    bLimitPosX := IPearlingMotorXYStatus.1,
    bLimitNegX := IPearlingMotorXYStatus.0,
    bHomeY := IPearlingMotorXYStatus.6,
    bLimitPosY := IPearlingMotorXYStatus.5,
    bLimitNegY := IPearlingMotorXYStatus.4,
    bHomeZ1 := IbPearlingHomeZ1,
    bLimitPosZ1 := IbPearlingPosLimitZ1,
    bLimitNegZ1 := IbPearlingNegLimitZ1,
    bHomeZ2 := IbPearlingHomeZ2,
    bLimitPosZ2 := IbPearlingPosLimitZ2,
    bLimitNegZ2 := IbPearlingNegLimitZ2,
    bChuck1Opened := IbPearlingChuck1Open,
    bChuck1Closed := IbPearlingChuck1Closed,
    bChuck2Opened := IbPearlingChuck2Open,
    bChuck2Closed := IbPearlingChuck2Closed,
    bResetErrors := sMMI_SyncVar.bResetErrors,
    bNewJob := sMMI_SyncVar.bNewJob,
    bStopReq := bStopRequest,
    bPauseReq := bPauseRequest,
    asStickData := asStickData,
    asStickDataMMI := asStickDataMMI,
    sStickDataShared := sStickDataShared,
    lrCompenseWeight1 := asStickDataMMI[0].iCompenseWeight,
    lrCompenseWeight2 := asStickDataMMI[1].iCompenseWeight,
    iComPort := C_COM_NUMBERS[CI_Pearling],
    sInTakeFromBarrel := sGiversTakers.sBarrelGiveToPearling,
    iContact1Distance := IPearlingContact1Distance,
    iContact2Distance := IPearlingContact2Distance,
    iLoadSensorValue := IPearlingWeightMeasure,
    eSharpenRunStatus := sRunData.sStatusSharpen,
    eBarrelRunStatus := sRunData.sStatusBarrel,
    eRunCommand := sRunData.eCmdPearling,
    bKeepBothHeadWarm := bPearlingHead1IsUsed AND bPearlingHead2IsUsed,
    eTableSideForLoader := eTableSideForLoader,
    sPartData := sMMI_ConfigFileData.sPartData,
    bHead1IsUsed := bPearlingHead1IsUsed,
    bHead2IsUsed := bPearlingHead2IsUsed,
    bParallelProduction := sMMI_ConfigFileData.bParallelProduction,
    iLeftVacuumFlow := aiTablePearlsVacuumFlow[PH_LEFT],
    iRightVacuumFlow := aiTablePearlsVacuumFlow[PH_RIGHT],
    iMachineWO := iMachineWO,
    iMachineSN := iMachineSN,
    yModulePosition := 0,
    sCurrentState := sMMI_SyncVar.sModPearling,
    TManualCmd := sMMI_ManualVar.TPearlingManual,
    sRecData := RxBuffer_MCR[CI_Pearling],
    sTransData := TxBuffer_MCR[CI_Pearling],
    asPearlData := sMMI_SyncVar.asPearlsData,
    sXAxisRef := TPearlingXAxis,
    sYAxisRef := TPearlingYAxis,
    sZ1AxisRef := TPearlingZ1Axis,
    sZ2AxisRef := TPearlingZ2Axis,
    sRunData := sRunData.TDataPearling,
    asProbingLog := sMMI_SyncVar.asProbingLog,
    bXAxisError => sMMI_SyncVar.abErrorsTable[ERR_PearlingAxisX],
    bYAxisError => sMMI_SyncVar.abErrorsTable[ERR_PearlingAxisY],
    bZ1AxisError => sMMI_SyncVar.abErrorsTable[ERR_PearlingAxisZ1],
    bZ2AxisError => sMMI_SyncVar.abErrorsTable[ERR_PearlingAxisZ2],
    bChuck1Error => sMMI_SyncVar.abErrorsTable[ERR_PearlingGripper1],
    bChuck2Error => sMMI_SyncVar.abErrorsTable[ERR_PearlingGripper2],
    bSpindle1Error => sMMI_SyncVar.abErrorsTable[ERR_PearlingSpindle1],
    bSpindle2Error => sMMI_SyncVar.abErrorsTable[ERR_PearlingSpindle2],
    bSecurityError => sMMI_SyncVar.abErrorsTable[ERR_PearlingSecurity],
    bMCRError => sMMI_SyncVar.abErrorsTable[ERR_PearlingMCR],
    bStick1Broken => sMMI_SyncVar.abErrorsTable[W_PearlingLeftStickBroken],
    bStick2Broken => sMMI_SyncVar.abErrorsTable[W_PearlingRightStickBroken],
    bStartPearlingMotor1 => QbPearlingStartMotor1,
    bStartPearlingMotor2 => QbPearlingStartMotor2,
    bOpenChuck1 => QbPearlingOpenChuck1,
    bOpenChuck2 => QbPearlingOpenChuck2,
    bActivateEject1 => QbPearlingActivateEject1,
    bActivateEject2 => QbPearlingActivateEject2,
    bActivateBlowing1 => QbPearlingActivateBlowing1,
    bActivateBlowing2 => QbPearlingActivateBlowing2,
    bAspirationPearling1On => bTableAspiration13On,
    bAspirationPearling2On => bTableAspiration24On,
    bAspirationSharpenOn => bSharpenAspirationOn,
    bStickContact1 => QbPearlingStickLed1,
    bStickContact2 => QbPearlingStickLed2,
    bCurrent1ReadError => sMMI_SyncVar.abErrorsTable[ERR_PearlingCurrent1],
    bCurrent2ReadError => sMMI_SyncVar.abErrorsTable[ERR_PearlingCurrent2],
    bMotor1Error => sMMI_SyncVar.abErrorsTable[ERR_PearlingMotor1],
    bMotor2Error => sMMI_SyncVar.abErrorsTable[ERR_PearlingMotor2],
    bPearlingWeight1OutOfToleranceError => sMMI_SyncVar.abErrorsTable[W_PearlingWeight1OutOfTolerance],
    bPearlingWeight2OutOfToleranceError => sMMI_SyncVar.abErrorsTable[W_PearlingWeight2OutOfTolerance],
    bStickNotTakenError => sMMI_SyncVar.abErrorsTable[ERR_BarrelStickNotTaken],
    bReady2ChangeTool => bPearlingReady4ChangeTool,
    iStickHead => iStickArea2Use,
    sOutTakeFromBarrel => sGiversTakers.sPearlingTakeFromBarrel,
    eSharpenRunCmd => sRunData.eCmdSharpen,
    eBarrelRunCmd => sRunData.eCmdBarrel,
    eRunStatus => sRunData.sStatusPearling,
    bManInterlockOut => bManInterlockPearling,
    adwMotorRunningHours => sMMI_SyncVar.sCounter.adwPearlingMotorRunningHours,
    adwSpindleRunningHours => sMMI_SyncVar.sCounter.adwPearlingSpindleRunningHours,
    bLeftSpindleUsedWarning => sMMI_SyncVar.abErrorsTable[W_PearlingLeftSpindleUsed],
    bRightSpindleUsedWarning => sMMI_SyncVar.abErrorsTable[W_PearlingRightSpindleUsed],
    bLeftMotorUsedWarning => sMMI_SyncVar.abErrorsTable[W_PearlingLeftMotorUsed],
    bRightMotorUsedWarning => sMMI_SyncVar.abErrorsTable[W_PearlingRightMotorUsed],
    bLeftSpindleLimitWarning => sMMI_SyncVar.abErrorsTable[W_PearlingLeftSpindleLimit],
    bRightSpindleLimitWarning => sMMI_SyncVar.abErrorsTable[W_PearlingRightSpindleLimit],
    bLeftSpindleHeatWarning => sMMI_SyncVar.abErrorsTable[W_PearlingLeftSpindleHeat],
    bRightSpindleHeatWarning => sMMI_SyncVar.abErrorsTable[W_PearlingRightSpindleHeat]); // PearlingHdl

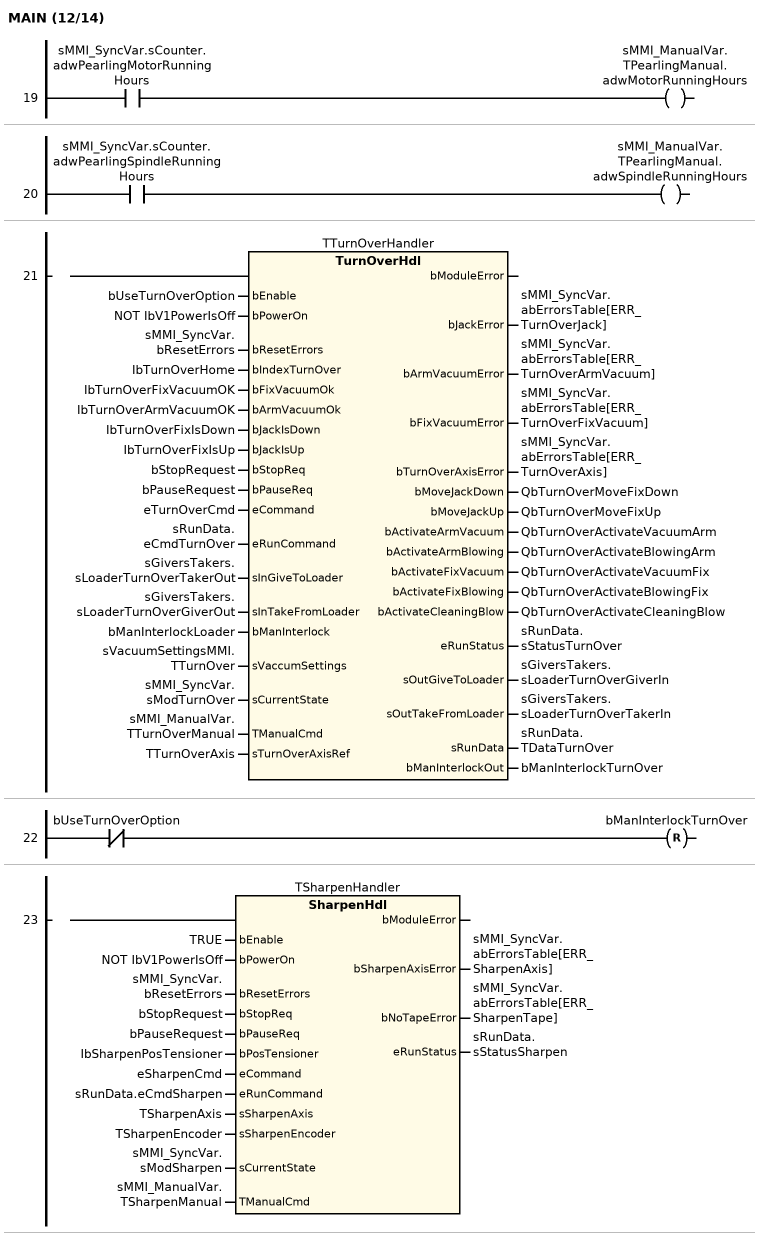
// NETWORK 19
sMMI_ManualVar.TPearlingManual.adwMotorRunningHours := sMMI_SyncVar.sCounter.adwPearlingMotorRunningHours;

// NETWORK 20
sMMI_ManualVar.TPearlingManual.adwSpindleRunningHours := sMMI_SyncVar.sCounter.adwPearlingSpindleRunningHours;

// NETWORK 21
TTurnOverHandler(
    bEnable := bUseTurnOverOption,
    bPowerOn := NOT IbV1PowerIsOff,
    bResetErrors := sMMI_SyncVar.bResetErrors,
    bIndexTurnOver := IbTurnOverHome,
    bFixVacuumOk := IbTurnOverFixVacuumOK,
    bArmVacuumOk := IbTurnOverArmVacuumOK,
    bJackIsDown := IbTurnOverFixIsDown,
    bJackIsUp := IbTurnOverFixIsUp,
    bStopReq := bStopRequest,
    bPauseReq := bPauseRequest,
    eCommand := eTurnOverCmd,
    eRunCommand := sRunData.eCmdTurnOver,
    sInGiveToLoader := sGiversTakers.sLoaderTurnOverTakerOut,
    sInTakeFromLoader := sGiversTakers.sLoaderTurnOverGiverOut,
    bManInterlock := bManInterlockLoader,
    sVaccumSettings := sVacuumSettingsMMI.TTurnOver,
    sCurrentState := sMMI_SyncVar.sModTurnOver,
    TManualCmd := sMMI_ManualVar.TTurnOverManual,
    sTurnOverAxisRef := TTurnOverAxis,
    bJackError => sMMI_SyncVar.abErrorsTable[ERR_TurnOverJack],
    bArmVacuumError => sMMI_SyncVar.abErrorsTable[ERR_TurnOverArmVacuum],
    bFixVacuumError => sMMI_SyncVar.abErrorsTable[ERR_TurnOverFixVacuum],
    bTurnOverAxisError => sMMI_SyncVar.abErrorsTable[ERR_TurnOverAxis],
    bMoveJackDown => QbTurnOverMoveFixDown,
    bMoveJackUp => QbTurnOverMoveFixUp,
    bActivateArmVacuum => QbTurnOverActivateVacuumArm,
    bActivateArmBlowing => QbTurnOverActivateBlowingArm,
    bActivateFixVacuum => QbTurnOverActivateVacuumFix,
    bActivateFixBlowing => QbTurnOverActivateBlowingFix,
    bActivateCleaningBlow => QbTurnOverActivateCleaningBlow,
    eRunStatus => sRunData.sStatusTurnOver,
    sOutGiveToLoader => sGiversTakers.sLoaderTurnOverGiverIn,
    sOutTakeFromLoader => sGiversTakers.sLoaderTurnOverTakerIn,
    sRunData => sRunData.TDataTurnOver,
    bManInterlockOut => bManInterlockTurnOver); // TurnOverHdl

// NETWORK 22
bManInterlockTurnOver R= NOT bUseTurnOverOption;

// NETWORK 23
TSharpenHandler(
    bEnable := TRUE,
    bPowerOn := NOT IbV1PowerIsOff,
    bResetErrors := sMMI_SyncVar.bResetErrors,
    bStopReq := bStopRequest,
    bPauseReq := bPauseRequest,
    bPosTensioner := IbSharpenPosTensioner,
    eCommand := eSharpenCmd,
    eRunCommand := sRunData.eCmdSharpen,
    sSharpenAxis := TSharpenAxis,
    sSharpenEncoder := TSharpenEncoder,
    sCurrentState := sMMI_SyncVar.sModSharpen,
    TManualCmd := sMMI_ManualVar.TSharpenManual,
    bSharpenAxisError => sMMI_SyncVar.abErrorsTable[ERR_SharpenAxis],
    bNoTapeError => sMMI_SyncVar.abErrorsTable[ERR_SharpenTape],
    eRunStatus => sRunData.sStatusSharpen); // SharpenHdl

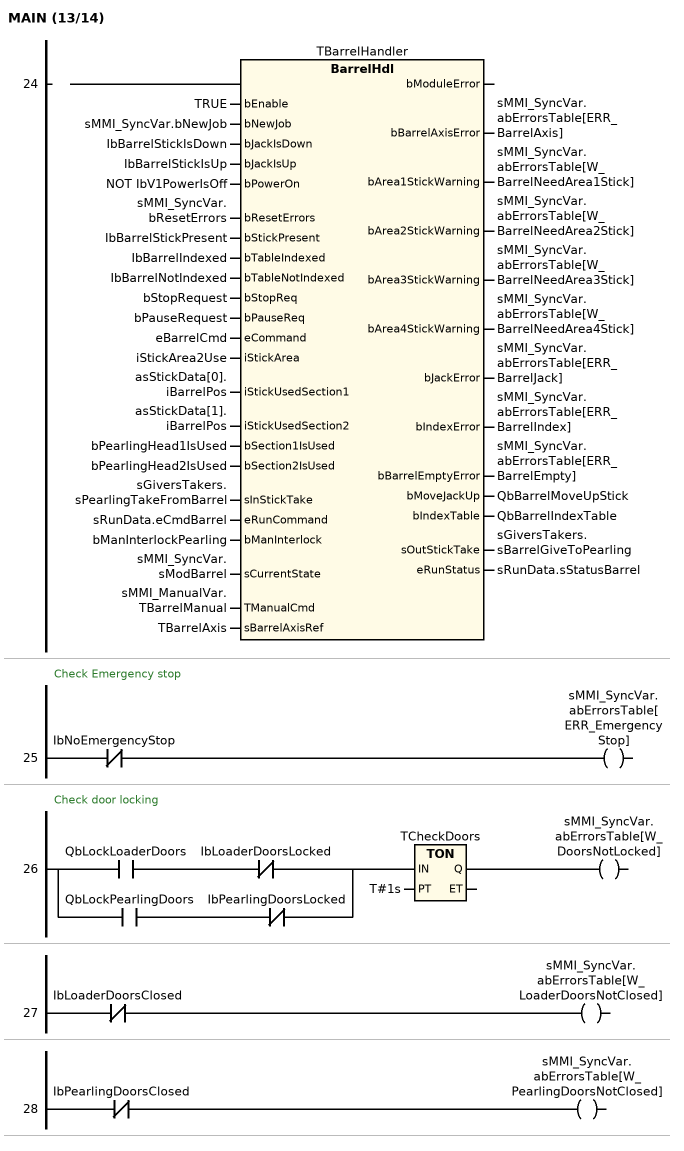
// NETWORK 24
TBarrelHandler(
    bEnable := TRUE,
    bNewJob := sMMI_SyncVar.bNewJob,
    bJackIsDown := IbBarrelStickIsDown,
    bJackIsUp := IbBarrelStickIsUp,
    bPowerOn := NOT IbV1PowerIsOff,
    bResetErrors := sMMI_SyncVar.bResetErrors,
    bStickPresent := IbBarrelStickPresent,
    bTableIndexed := IbBarrelIndexed,
    bTableNotIndexed := IbBarrelNotIndexed,
    bStopReq := bStopRequest,
    bPauseReq := bPauseRequest,
    eCommand := eBarrelCmd,
    iStickArea := iStickArea2Use,
    iStickUsedSection1 := asStickData[0].iBarrelPos,
    iStickUsedSection2 := asStickData[1].iBarrelPos,
    bSection1IsUsed := bPearlingHead1IsUsed,
    bSection2IsUsed := bPearlingHead2IsUsed,
    sInStickTake := sGiversTakers.sPearlingTakeFromBarrel,
    eRunCommand := sRunData.eCmdBarrel,
    bManInterlock := bManInterlockPearling,
    sCurrentState := sMMI_SyncVar.sModBarrel,
    TManualCmd := sMMI_ManualVar.TBarrelManual,
    sBarrelAxisRef := TBarrelAxis,
    bBarrelAxisError => sMMI_SyncVar.abErrorsTable[ERR_BarrelAxis],
    bArea1StickWarning => sMMI_SyncVar.abErrorsTable[W_BarrelNeedArea1Stick],
    bArea2StickWarning => sMMI_SyncVar.abErrorsTable[W_BarrelNeedArea2Stick],
    bArea3StickWarning => sMMI_SyncVar.abErrorsTable[W_BarrelNeedArea3Stick],
    bArea4StickWarning => sMMI_SyncVar.abErrorsTable[W_BarrelNeedArea4Stick],
    bJackError => sMMI_SyncVar.abErrorsTable[ERR_BarrelJack],
    bIndexError => sMMI_SyncVar.abErrorsTable[ERR_BarrelIndex],
    bBarrelEmptyError => sMMI_SyncVar.abErrorsTable[ERR_BarrelEmpty],
    bMoveJackUp => QbBarrelMoveUpStick,
    bIndexTable => QbBarrelIndexTable,
    sOutStickTake => sGiversTakers.sBarrelGiveToPearling,
    eRunStatus => sRunData.sStatusBarrel); // BarrelHdl

// NETWORK 25
// Check Emergency stop
sMMI_SyncVar.abErrorsTable[ERR_EmergencyStop] := NOT IbNoEmergencyStop;

// NETWORK 26
// Check door locking
TCheckDoors(IN := QbLockLoaderDoors AND NOT IbLoaderDoorsLocked OR QbLockPearlingDoors AND NOT IbPearlingDoorsLocked, PT := T#1s); // TON
sMMI_SyncVar.abErrorsTable[W_DoorsNotLocked] := TCheckDoors.Q;

// NETWORK 27
sMMI_SyncVar.abErrorsTable[W_LoaderDoorsNotClosed] := NOT IbLoaderDoorsClosed;

// NETWORK 28
sMMI_SyncVar.abErrorsTable[W_PearlingDoorsNotClosed] := NOT IbPearlingDoorsClosed;

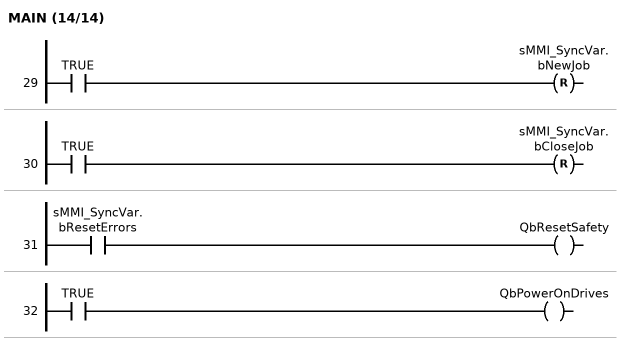
// NETWORK 29
sMMI_SyncVar.bNewJob R= TRUE;

// NETWORK 30
sMMI_SyncVar.bCloseJob R= TRUE;

// NETWORK 31
QbResetSafety := sMMI_SyncVar.bResetErrors;

// NETWORK 32
QbPowerOnDrives := TRUE;

END_PROGRAM

// ---- POUs/Manager/Manager.TcPOU
FUNCTION_BLOCK Manager
VAR_INPUT
	bEnable						: BOOL;
	bPowerOn					: BOOL;
	bNewJob						: BOOL;
	bEndOfJob					: BOOL;
	sMachineData				: TMachineData;
	bNoEmergencyStop			: BOOL;
	bLoaderDoorsLocked			: BOOL;
	bPearlingDoorsLocked		: BOOL;
	bLoaderDoorsClosed			: BOOL;
	bPearlingDoorsClosed			: BOOL;
	bChangeToolReq				: BOOL;
	sProdLot						: TProductionLot;
	sConfigFileData				: TConfigFileData;
	bSimPearling					: BOOL;
	dwStartJobElapsedTime		: DWORD;
	bVisionInConfig				: BOOL;
	bFillMDE						: BOOL;
	bDisableCleanAfterPearling		: BOOL;
END_VAR
VAR_OUTPUT
	bModuleError					: BOOL;
	bGreenLight					: BOOL;
	bRedLight					: BOOL;
	bBlueLight					: BOOL;
	bOrangeLight					: BOOL;
	bLockLoaderDoors			: BOOL;
	bLockPearlingDoors			: BOOL;
	bCanChangeTool				: BOOL;
	eCmdLoader					: TModuleCommands;
	eCmdTable					: TModuleCommands;
	eCmdPearling				: TModuleCommands;
	eCmdTurnOver				: TModuleCommands;
	eCmdBarrel					: TModuleCommands;
	eCmdSharpen				: TModuleCommands;
	eCmdLift1					: TModuleCommands;
	eCmdLift2					: TModuleCommands;
	eCmdReject					: TModuleCommands;
	eCmdVision					: TModuleCommands;
	eCmdUtilities					: TModuleCommands;
	bPearlingHead1IsUsed		: BOOL;
	bPearlingHead2IsUsed		: BOOL;
	bMMIEmergencyStop			: BOOL;
	bMMIDoorsPearling			: BOOL;
	bMMIDoorsLoader			: BOOL;
	bStopRequest				: BOOL;
	bPauseRequest				: BOOL;
	bReadyForChangeJob			: BOOL;
	bLayeringWithTwoParts		: BOOL;
	eManagerRunStep			: TModuleSteps;
	bJobInProgress				: BOOL 				:= FALSE;
	TJobElapsed					: TIME;
	dwProdEstimatedTimeLeft		: DWORD;
	dwMeanMTBF				: DWORD;
	bConfigError					: BOOL;
	dwMachineOnHours			: DWORD;
	TInProdHours				: DWORD;
END_VAR
VAR_IN_OUT
	eMachineMode				: TMachineMode;
	sModeMask					: TMachineModeMask;
	sModeReq					: TMachineModeMask;
	sMachineSafetyCmd			: TMachineManual;
	bResetErrors					: BOOL;
	bPurgeReq					: BOOL;
	sRunData					: TRunData;
	bSavePersistent				: BOOL;
	bResetMTBF					: BOOL;
	sDashboardCmd				: TDashboardCmd;
	sProductionCmd				: TProductionCmd;
END_VAR
VAR PERSISTENT
	TMaxStopppingTime			: TIME := t#4m;
	TMaxPausingTime			: TIME := t#5s;
	iMTBFCounter				: INT;
	dwMTBFTotalTime			: DWORD;
END_VAR
VAR CONSTANT
	 iMaxModule					: INT := 10;
END_VAR
VAR
	bRunTestMode				: BOOL					 := FALSE;
	bInError						: BOOL;
	bInWarning					: BOOL;
	TForceStop					: TON;
	TReadyToStopTimer			: TON;
	TTapReset					: TON;
	TCheckErrors					: HandleErrors;
	TBlinking					: TBlink;
	bBlinking						: BOOL;
	eStep						: TModuleSteps := SP_RunStp0;
	bAllowDoorsControl			: BOOL;
	eLastMachineMode			: TMachineMode;
	bOneModuleInStop			: BOOL;
	bOneModuleInReady			: BOOL;
	bAllModuleInReady			: BOOL;
	bAllModuleInStop				: BOOL;
	bAllModuleInPause			: BOOL;
	bOneModuleInReadyOrStop	: BOOL;
	bAllModuleInReadyOrStop		: BOOL;
	bOneModuleInPause			: BOOL;
	aTModuleStatus				: ARRAY[0..iMaxModule] OF TModuleStatus;
	i							: INT;
	eCmdAll						: TModuleCommands;
	TManagerDashboard			: ManagerDashboard;
	TManagerRun				: ManagerRun;
	TManagerRunTest			: ManagerRunTest;
	bRunInit						: BOOL;
	bNewJobForRun				: BOOL;
	bDoChangeTool				: BOOL;
	bDoInitAfterStop				: BOOL;
	TWritePersistentData			: FB_WritePersistentData;
	TJobElapsedCounter			: StopWatch;
	TMTBFCounter				: MTBFCounter;
	dwJobQty					: DWORD;
	bInJobMode					: BOOL;
	bComputeMTBF				: BOOL						:= FALSE;
	iMDEAlarm					: INT;
	TMachineOnCounter			: RunningCounter;
	TInProdCounter				: RunningCounter;
	bResetMachineCounters		: BOOL						:= FALSE;
END_VAR

(* Reset errors delay*)
TTapReset(IN := bResetErrors,PT := t#100ms);
IF TTapReset.Q THEN
	bResetErrors := FALSE;
END_IF


(* Handle doors locking *)
IF bAllowDoorsControl THEN
	sMachineSafetyCmd.bCanLockDoor := NOT (bLoaderDoorsLocked AND bPearlingDoorsLocked);
	sMachineSafetyCmd.bCanUnlockDoor := bLockLoaderDoors OR bLockPearlingDoors; (*NOT sMachineSafetyCmd.bCanLockDoor;*)
	IF sMachineSafetyCmd.bLockDoor THEN
		bLockLoaderDoors := TRUE;
		bLockPearlingDoors := TRUE;
		sMachineSafetyCmd.bLockDoor := FALSE;
	END_IF
	IF sMachineSafetyCmd.bUnlockDoor THEN
		bLockLoaderDoors := FALSE;
		bLockPearlingDoors := FALSE;
		sMachineSafetyCmd.bUnlockDoor := FALSE;
	END_IF
	IF NOT bNoEmergencyStop THEN
		bLockLoaderDoors := FALSE;
		bLockPearlingDoors := FALSE;
	END_IF
ELSE
	sMachineSafetyCmd.bCanLockDoor := FALSE;
	sMachineSafetyCmd.bLockDoor := FALSE;
	sMachineSafetyCmd.bCanUnlockDoor := FALSE;
	sMachineSafetyCmd.bUnlockDoor := FALSE;
	(* Lock doors *)
	bLockLoaderDoors := TRUE;
	bLockPearlingDoors := TRUE;
END_IF

bMMIEmergencyStop := NOT bNoEmergencyStop;
bMMIDoorsPearling := NOT bPearlingDoorsLocked OR NOT bPearlingDoorsClosed;
bMMIDoorsLoader := NOT bLoaderDoorsLocked OR NOT bLoaderDoorsClosed ;

(* Create blinking *)
TBlinking(
	bEnable			:= TRUE,
	tOnPeriod		:= t#500ms,
	tOffPeriod		:= t#500ms,
	bBlink			=> bBlinking
);

(* Check error or warning state *)
TCheckErrors(
	bEnable			:= TRUE,
	abErrorsTable	:= sMachineData.abErrorsTable,
	bInError			=> bInError,
	bInWarning		=> bInWarning,
	iMDEAlarm		=> iMDEAlarm
);

(* Update lights *)
bGreenLight := (eMachineMode = MM_Running) OR (eMachineMode = MM_Purging) OR
		((eMachineMode <> MM_Stopped) AND (eMachineMode <> MM_Ready) AND bBlinking);
bRedLight := bInError;
bBlueLight := bInWarning;
bOrangeLight := NOT (bLoaderDoorsLocked AND bPearlingDoorsLocked);

(* Clear commands on modules *)
eCmdLoader := MC_NoCmd;
eCmdTable:= MC_NoCmd;
eCmdPearling := MC_NoCmd;
eCmdTurnOver := MC_NoCmd;
eCmdBarrel := MC_NoCmd;
eCmdSharpen := MC_NoCmd;
eCmdLift1 := MC_NoCmd;
eCmdLift2 := MC_NoCmd;
eCmdReject := MC_NoCmd;
eCmdVision := MC_NoCmd;
eCmdUtilities := MC_NoCmd;
eCmdAll := MC_NoCmd;

aTModuleStatus[0] := sMachineData.sModLoader.eStatus;
aTModuleStatus[1] := sMachineData.sModPearling.eStatus;
aTModuleStatus[2] := sMachineData.sModTable.eStatus;
aTModuleStatus[3] := sMachineData.sModTurnOver.eStatus;
aTModuleStatus[4] := sMachineData.sModBarrel.eStatus;
aTModuleStatus[5] := sMachineData.sModSharpen.eStatus;
aTModuleStatus[6] := sMachineData.sModLift1.eStatus;
aTModuleStatus[7] := sMachineData.sModLift2.eStatus;
aTModuleStatus[8] := sMachineData.sModReject.eStatus;
aTModuleStatus[9] := sMachineData.sModVision.eStatus;
aTModuleStatus[10] := sMachineData.sModUtilities.eStatus;

bOneModuleInStop := FALSE;
bOneModuleInReady := FALSE;
bOneModuleInPause := FALSE;
bAllModuleInReady := TRUE;
bAllModuleInPause := TRUE;
bAllModuleInReadyOrStop := TRUE;
bAllModuleInStop := TRUE;
FOR i:=0 TO iMaxModule DO
	IF aTModuleStatus[i] = MS_Paused THEN bOneModuleInPause := TRUE; END_IF
	IF aTModuleStatus[i] = MS_Stopped THEN bOneModuleInStop := TRUE; END_IF
	IF aTModuleStatus[i] = MS_Ready THEN bOneModuleInReady := TRUE; END_IF
	IF aTModuleStatus[i] <> MS_Paused THEN bAllModuleInPause := FALSE; END_IF
	IF aTModuleStatus[i] <> MS_Ready THEN bAllModuleInReady := FALSE; END_IF
	IF aTModuleStatus[i] <> MS_Stopped THEN bAllModuleInStop := FALSE; END_IF
	IF aTModuleStatus[i] <> MS_Ready AND aTModuleStatus[i] <> MS_Stopped THEN bAllModuleInReadyOrStop := FALSE; END_IF
END_FOR
bOneModuleInReadyOrStop := bOneModuleInStop OR bOneModuleInReady;

IF (eMachineMode <> eLastMachineMode) THEN
	eStep := SP_RunStp0;
	eLastMachineMode := eMachineMode;
END_IF

